// TwinCAT 3 PLC project PRG_MachineSystem
// ProgramVersion: 3.1.4024.0
// CompilerDefines: VISU_USEWSTRING
// libraries:
//   B_Base, * (RafalOS)
//   B_Base_HMI_Connector, * (RafalOS)
//   B_HMIManager, * (RafałOS)
//   B_MachineControl, * (RafalOS)
//   B_MachineControl_HMI_Connector, * (RafalOS)
//   B_MachineSystem, * (RafalOS)
//   B_PLCHMIManager, * (RafalOS)
//   Tc2_Standard, * (Beckhoff Automation GmbH)
//   Tc2_System, * (Beckhoff Automation GmbH)
//   Tc3_Module, * (Beckhoff Automation GmbH)
//   VisuSymbols,3.5.10.0,System
// project tree:
//   / DefaultInit.TcTTO, GlobalTextList.TcGTLO, MachineInit.TcTTO, PlcTask.TcTTO (not stored), Visualization Manager.TcVMO (not stored), VISU_TASK.TcTTO (not stored)
//   GVLs/ GVL_MachineVariable.TcGVL, GVL_TE1.TcGVL, GVL_TE2.TcGVL
//   POUs/01_MachineConfiguration/ FB_MachineConfiguration.TcPOU
//   POUs/02_HMIConfiguration/ FB_HMIConfiguration.TcPOU
//   POUs/03_CreatingTemplateRecipe/ FB_MachineTemplate1.TcPOU, FB_MachineTemplate2.TcPOU, FB_MachineTemplate3.TcPOU
//   POUs/04_TopElement1/3GE_B/ FB_GroupE_TE1.TcPOU, ITF_GroupE_TE1.TcIO, ITF_GroupE_TE1_HMI_Connector.TcIO, ITF_GroupE_TE1_HMI_Init.TcIO
//   POUs/04_TopElement1/3GE_B_HMI/ FB_GroupE_TE1_HMI.TcPOU, ITF_GroupE_TE1_HMI.TcIO, ST_GroupE_TE1_HMI.TcDUT, ST_GroupE_TE1_HMI_Link.TcDUT
//   POUs/04_TopElement1/9TE_B/ FB_TopElement1.TcPOU, ITF_TopElement1_HMI_Init.TcIO, ITF_TopElement1_HMI_Connector.TcIO, ITF_TopElement1.TcIO (not stored)
//   POUs/04_TopElement1/9TE_B_HMI/ FB_TopElement1_HMI.TcPOU, ITF_TopElement1_HMI.TcIO, ST_TopElement1_HMI.TcDUT, ST_TopElement1_HMI_Link.TcDUT
//   POUs/04_TopElement1/1C_B/ FB_Component_TE1.TcPOU, ITF_Component_TE1.TcIO, ITF_Component_TE1_HMI_Init.TcIO, ITF_Component_TE1_HMI_Connector.TcIO
//   POUs/04_TopElement1/2CE_B/ FB_ControlE_TE1.TcPOU, ITF_ControlE_TE1.TcIO, ITF_ControlE_TE1_HMI_Connector.TcIO, ITF_ControlE_TE1_HMI_Init.TcIO
//   POUs/04_TopElement1/1C_B_HMI/ FB_Component_TE1_HMI.TcPOU, ITF_Component_TE1_HMI.TcIO, ST_Component_TE1_HMI.TcDUT, ST_Component_TE1_HMI_Link.TcDUT
//   POUs/04_TopElement1/2CE_B_HMI/ FB_ControlE_TE1_HMI.TcPOU, ITF_ControlE_TE1_HMI.TcIO, ST_ControlE_TE1_HMI.TcDUT, ST_ControlE_TE1_HMI_Link.TcDUT
//   POUs/05_TopElement2/1C_B/ FB_Component_TE2.TcPOU, ITF_Component_TE2.TcIO, ITF_Component_TE2_HMI_Connector.TcIO, ITF_Component_TE2_HMI_Init.TcIO
//   POUs/05_TopElement2/1C_B_HMI/ FB_Component_TE2_HMI.TcPOU, ITF_Component_TE2_HMI.TcIO, ST_Component_TE2_HMI.TcDUT, ST_Component_TE2_HMI_Link.TcDUT
//   POUs/05_TopElement2/2CE_B/ FB_ControlE_TE2.TcPOU, ITF_ControlE_TE2.TcIO, ITF_ControlE_TE2_HMI_Connector.TcIO, ITF_ControlE_TE2_HMI_Init.TcIO
//   POUs/05_TopElement2/2CE_B_HMI/ FB_ControlE_TE2_HMI.TcPOU, ITF_ControlE_TE2_HMI.TcIO, ST_ControlE_TE2_HMI.TcDUT, ST_ControlE_TE2_HMI_Link.TcDUT
//   POUs/05_TopElement2/3GE_B/ FB_GroupE_TE2.TcPOU, ITF_GroupE_TE2.TcIO, ITF_GroupE_TE2_HMI_Connector.TcIO, ITF_GroupE_TE2_HMI_Init.TcIO
//   POUs/05_TopElement2/3GE_B_HMI/ FB_GroupE_TE2_HMI.TcPOU, ITF_GroupE_TE2_HMI.TcIO, ST_GroupE_TE2_HMI.TcDUT, ST_GroupE_TE2_HMI_Link.TcDUT
//   POUs/05_TopElement2/9TE_B/ FB_TopElement2.TcPOU, ITF_TopElement2.TcIO, ITF_TopElement2_HMI_Connector.TcIO, ITF_TopElement2_HMI_Init.TcIO
//   POUs/05_TopElement2/9TE_B_HMI/ FB_TopElement2_HMI.TcPOU, ITF_TopElement2_HMI.TcIO, ST_TopElement2_HMI.TcDUT, ST_TopElement2_HMI_Link.TcDUT
//   POUs/ PRG_MachineConfigure.TcPOU
//   VISUs/ MainScreen.TcVIS
// real-time tasks:
//   TASK PlcTask: cycle T#10ms, priority 10, ADS port 350
//   TASK VISU_TASK: cycle T#200000us, priority 12, ADS port 351
//   TASK DefaultInit: cycle T#10ms, priority 20, ADS port 352
//   TASK MachineInit: cycle T#10ms, priority 21, ADS port 353

CONFIGURATION PRG_MachineSystem
    RESOURCE PLC ON TwinCAT3
        TASK DefaultInit(INTERVAL := T#10ms, PRIORITY := 20);
        TASK MachineInit(INTERVAL := T#10ms, PRIORITY := 21);
        PROGRAM PRG_SystemControlMachineInit WITH DefaultInit : PRG_SystemControlMachineInit;
        PROGRAM PRG_ControlHMIInit WITH DefaultInit : PRG_ControlHMIInit;
        PROGRAM PRG_MachineConfigure WITH MachineInit : PRG_MachineConfigure;
    END_RESOURCE
END_CONFIGURATION

// ---- POUs/04_TopElement1/3GE_B_HMI/ST_GroupE_TE1_HMI.TcDUT
TYPE ST_GroupE_TE1_HMI :
STRUCT
	bZmienneTypoweDlaGE_TE1	: BOOL;
	
END_STRUCT
END_TYPE

// ---- POUs/04_TopElement1/3GE_B_HMI/ST_GroupE_TE1_HMI_Link.TcDUT
TYPE ST_GroupE_TE1_HMI_Link EXTENDS ST_BaseGroupElement_HMI_Link :
STRUCT
	stGroupE_TE1		: ST_GroupE_TE1_HMI;
	
	stControlE1_TE1		: ST_ControlE_TE1_HMI_Link;
	stControlE2_TE1		: ST_ControlE_TE1_HMI_Link;
	
	stComponetE1_TE1	: ST_Component_TE1_HMI_Link;
	stComponetE2_TE1	: ST_Component_TE1_HMI_Link;
	stComponetE3_TE1	: ST_Component_TE1_HMI_Link;
	stComponetE4_TE1	: ST_Component_TE1_HMI_Link;
	
END_STRUCT
END_TYPE

// ---- POUs/04_TopElement1/9TE_B_HMI/ST_TopElement1_HMI.TcDUT
TYPE ST_TopElement1_HMI :
STRUCT
	bZmienneTypoweDlaTopElement1	: BOOL;
	
END_STRUCT
END_TYPE

// ---- POUs/04_TopElement1/9TE_B_HMI/ST_TopElement1_HMI_Link.TcDUT
TYPE ST_TopElement1_HMI_Link EXTENDS ST_BaseTopElement_HMI_Link :
STRUCT
	stTopElement		: ST_TopElement1_HMI;
	
	stGE1				: ST_GroupE_TE1_HMI_Link;
	
	stCE1				: ST_ControlE_TE1_HMI_Link;
	stCE2				: ST_ControlE_TE1_HMI_Link;
	
	stC1				: ST_Component_TE1_HMI_Link;
	stC2				: ST_Component_TE1_HMI_Link;
	stC3				: ST_Component_TE1_HMI_Link;
	
END_STRUCT
END_TYPE

// ---- POUs/04_TopElement1/1C_B_HMI/ST_Component_TE1_HMI.TcDUT
TYPE ST_Component_TE1_HMI :
STRUCT
	bZmienneTypoweDlaComponent_TE1	: BOOL;
	
END_STRUCT
END_TYPE

// ---- POUs/04_TopElement1/1C_B_HMI/ST_Component_TE1_HMI_Link.TcDUT
TYPE ST_Component_TE1_HMI_Link EXTENDS ST_BaseComponent_HMI_Link :
STRUCT
	stComponent_TE1		: ST_Component_TE1_HMI;
	
	
END_STRUCT
END_TYPE

// ---- POUs/04_TopElement1/2CE_B_HMI/ST_ControlE_TE1_HMI.TcDUT
TYPE ST_ControlE_TE1_HMI :
STRUCT
	bZmienneTypoweDlaCE_TE1	: BOOL;
	
END_STRUCT
END_TYPE

// ---- POUs/04_TopElement1/2CE_B_HMI/ST_ControlE_TE1_HMI_Link.TcDUT
TYPE ST_ControlE_TE1_HMI_Link EXTENDS ST_BaseControlElement_HMI_Link :
STRUCT
	stControlE_TE1		: ST_ControlE_TE1_HMI;
	
	stComponetE1_TE1	: ST_Component_TE1_HMI_Link;
	stComponetE2_TE1	: ST_Component_TE1_HMI_Link;
	stComponetE3_TE1	: ST_Component_TE1_HMI_Link;
	stComponetE4_TE1	: ST_Component_TE1_HMI_Link;
	
END_STRUCT
END_TYPE

// ---- POUs/05_TopElement2/1C_B_HMI/ST_Component_TE2_HMI.TcDUT
TYPE ST_Component_TE2_HMI :
STRUCT
	bZmienneTypoweDlaComponent_TE2	: BOOL;
	
END_STRUCT
END_TYPE

// ---- POUs/05_TopElement2/1C_B_HMI/ST_Component_TE2_HMI_Link.TcDUT
TYPE ST_Component_TE2_HMI_Link EXTENDS ST_BaseComponent_HMI_Link :
STRUCT
	stComponent_TE2		: ST_Component_TE2_HMI;
	
	
END_STRUCT
END_TYPE

// ---- POUs/05_TopElement2/2CE_B_HMI/ST_ControlE_TE2_HMI.TcDUT
TYPE ST_ControlE_TE2_HMI :
STRUCT
	bZmienneTypoweDlaCE_TE2	: BOOL;
	
END_STRUCT
END_TYPE

// ---- POUs/05_TopElement2/2CE_B_HMI/ST_ControlE_TE2_HMI_Link.TcDUT
TYPE ST_ControlE_TE2_HMI_Link EXTENDS ST_BaseControlElement_HMI_Link :
STRUCT
	stControlE_TE2		: ST_ControlE_TE2_HMI;
	
	stComponetE1_TE2	: ST_Component_TE2_HMI_Link;
	stComponetE2_TE2	: ST_Component_TE2_HMI_Link;
	stComponetE3_TE2	: ST_Component_TE2_HMI_Link;
	stComponetE4_TE2	: ST_Component_TE2_HMI_Link;
	
END_STRUCT
END_TYPE

// ---- POUs/05_TopElement2/3GE_B_HMI/ST_GroupE_TE2_HMI.TcDUT
TYPE ST_GroupE_TE2_HMI :
STRUCT
	bZmienneTypoweDlaGE_TE2	: BOOL;
	
END_STRUCT
END_TYPE

// ---- POUs/05_TopElement2/3GE_B_HMI/ST_GroupE_TE2_HMI_Link.TcDUT
TYPE ST_GroupE_TE2_HMI_Link EXTENDS ST_BaseGroupElement_HMI_Link :
STRUCT
	stGroupE_TE2		: ST_GroupE_TE2_HMI;
	
	stControlE1_TE2		: ST_ControlE_TE2_HMI_Link;
	stControlE2_TE2		: ST_ControlE_TE2_HMI_Link;
	
	stComponetE1_TE2	: ST_Component_TE2_HMI_Link;
	stComponetE2_TE2	: ST_Component_TE2_HMI_Link;
	stComponetE3_TE2	: ST_Component_TE2_HMI_Link;
	stComponetE4_TE2	: ST_Component_TE2_HMI_Link;
	
END_STRUCT
END_TYPE

// ---- POUs/05_TopElement2/9TE_B_HMI/ST_TopElement2_HMI.TcDUT
TYPE ST_TopElement2_HMI :
STRUCT
	bZmienneTypoweDlaTopElement2	: BOOL;
	
END_STRUCT
END_TYPE

// ---- POUs/05_TopElement2/9TE_B_HMI/ST_TopElement2_HMI_Link.TcDUT
TYPE ST_TopElement2_HMI_Link EXTENDS ST_BaseTopElement_HMI_Link :
STRUCT
	stTopElement		: ST_TopElement2_HMI;
	
	stGE1				: ST_GroupE_TE2_HMI_Link;
	
	stCE1				: ST_ControlE_TE2_HMI_Link;
	stCE2				: ST_ControlE_TE2_HMI_Link;
	
	stC1				: ST_Component_TE2_HMI_Link;
	stC2				: ST_Component_TE2_HMI_Link;
	stC3				: ST_Component_TE2_HMI_Link;
	
END_STRUCT
END_TYPE

// ---- GVLs/GVL_MachineVariable.TcGVL
{attribute 'qualified_only'}
VAR_GLOBAL
	fbMachineConfiguration		: FB_MachineConfiguration;
	fbHMIConfiguration			: FB_HMIConfiguration;
	
	fbMachineTemplate1			: FB_MachineTemplate1;
	fbMachineTemplate2			: FB_MachineTemplate2;
	fbMachineTemplate3			: FB_MachineTemplate3;
	
END_VAR

// ---- GVLs/GVL_TE1.TcGVL
{attribute 'qualified_only'}
VAR_GLOBAL
(*	Control Element dla top element	*)
	fbComponent1CE1_TE1		: FB_Component_TE1;
	fbComponent2CE1_TE1		: FB_Component_TE1;
	fbComponent3CE1_TE1		: FB_Component_TE1;
	fbComponent4CE1_TE1		: FB_Component_TE1;
		
	fbControlE1_TE1			: FB_ControlE_TE1 (
								itfC1										:= fbComponent1CE1_TE1,
	                            itfC2										:= fbComponent2CE1_TE1,
	                            itfC3										:= fbComponent3CE1_TE1,
	                            itfC4										:= fbComponent4CE1_TE1
							);

	fbComponent1CE2_TE1		: FB_Component_TE1;
	fbComponent2CE2_TE1		: FB_Component_TE1;
	fbComponent3CE2_TE1		: FB_Component_TE1;
	fbComponent4CE2_TE1		: FB_Component_TE1;
		
	fbControlE2_TE1			: FB_ControlE_TE1 (
								itfC1										:= fbComponent1CE2_TE1,
	                            itfC2										:= fbComponent2CE2_TE1,
	                            itfC3										:= fbComponent3CE2_TE1,
	                            itfC4										:= fbComponent4CE2_TE1
							);
							
(*	element złożony	*)
	fbComponent1GE1_TE1			: FB_Component_TE1;
	fbComponent2GE1_TE1			: FB_Component_TE1;
	fbComponent3GE1_TE1			: FB_Component_TE1;
	fbComponent4GE1_TE1			: FB_Component_TE1;

	fbComponent1CE1GE1_TE1		: FB_Component_TE1;
	fbComponent2CE1GE1_TE1		: FB_Component_TE1;
	fbComponent3CE1GE1_TE1		: FB_Component_TE1;
	fbComponent4CE1GE1_TE1		: FB_Component_TE1;
		
	fbControlE1GE1_TE1			: FB_ControlE_TE1 (
								itfC1										:= fbComponent1CE1GE1_TE1,
	                            itfC2										:= fbComponent2CE1GE1_TE1,
	                            itfC3										:= fbComponent3CE1GE1_TE1,
	                            itfC4										:= fbComponent4CE1GE1_TE1
							);

	fbComponent1CE2GE1_TE1		: FB_Component_TE1;
	fbComponent2CE2GE1_TE1		: FB_Component_TE1;
	fbComponent3CE2GE1_TE1		: FB_Component_TE1;
	fbComponent4CE2GE1_TE1		: FB_Component_TE1;
		
	fbControlE2GE1_TE1			: FB_ControlE_TE1 (
								itfC1										:= fbComponent1CE2GE1_TE1,
	                            itfC2										:= fbComponent2CE2GE1_TE1,
	                            itfC3										:= fbComponent3CE2GE1_TE1,
	                            itfC4										:= fbComponent4CE2GE1_TE1
							);

	fbGroupE1_TE1			: FB_GroupE_TE1 (
								itfCE1										:= fbControlE1GE1_TE1,
	                            itfCE2										:= fbControlE2GE1_TE1,
	                            itfC1										:= fbComponent1GE1_TE1,
	                            itfC2										:= fbComponent2GE1_TE1,
	                            itfC3										:= fbComponent3GE1_TE1,
	                            itfC4										:= fbComponent4GE1_TE1
							);
							
							
(*	Komponenty TopElement1	*)
	fbComponent1_TE1		: FB_Component_TE1;
	fbComponent2_TE1		: FB_Component_TE1;
	fbComponent3_TE1		: FB_Component_TE1;
	
	fbTopElement1			: FB_TopElement1 (
								itfGE1										:= fbGroupE1_TE1,
								itfCE1										:= fbControlE1_TE1,
	                            itfCE2										:= fbControlE2_TE1,
								itfC1										:= fbComponent1_TE1,
								itfC2										:= fbComponent2_TE1,
								itfC3										:= fbComponent3_TE1
							);
	
(*	HMI	*)
	(* controlelementy *)
	fbComponent1CE1_TE1_HMI	: FB_Component_TE1_HMI (
								itfBaseLoggerConnector						:= GVL_SystemVariable.fbLogger,
	                            itfComponent_TE1Connector					:= fbComponent1CE1_TE1
							);
	fbComponent2CE1_TE1_HMI	: FB_Component_TE1_HMI (
								itfBaseLoggerConnector						:= GVL_SystemVariable.fbLogger,
	                            itfComponent_TE1Connector					:= fbComponent2CE1_TE1
							);
	fbComponent3CE1_TE1_HMI	: FB_Component_TE1_HMI (
								itfBaseLoggerConnector						:= GVL_SystemVariable.fbLogger,
	                            itfComponent_TE1Connector					:= fbComponent3CE1_TE1
							);
	fbComponent4CE1_TE1_HMI	: FB_Component_TE1_HMI (
								itfBaseLoggerConnector						:= GVL_SystemVariable.fbLogger,
	                            itfComponent_TE1Connector					:= fbComponent4CE1_TE1
							);

	fbControlE1_TE1_HMI			: FB_ControlE_TE1_HMI (
								itfBaseLoggerConnector						:= GVL_SystemVariable.fbLogger,
								itfControlE_TE1Connector					:= fbControlE1_TE1,
								itfC1										:= fbComponent1CE1_TE1_HMI,
	                            itfC2										:= fbComponent2CE1_TE1_HMI,
	                            itfC3										:= fbComponent3CE1_TE1_HMI,
	                            itfC4										:= fbComponent4CE1_TE1_HMI
							);

	fbComponent1CE2_TE1_HMI	: FB_Component_TE1_HMI (
								itfBaseLoggerConnector						:= GVL_SystemVariable.fbLogger,
	                            itfComponent_TE1Connector					:= fbComponent1CE2_TE1
							);
	fbComponent2CE2_TE1_HMI	: FB_Component_TE1_HMI (
								itfBaseLoggerConnector						:= GVL_SystemVariable.fbLogger,
	                            itfComponent_TE1Connector					:= fbComponent2CE2_TE1
							);
	fbComponent3CE2_TE1_HMI	: FB_Component_TE1_HMI (
								itfBaseLoggerConnector						:= GVL_SystemVariable.fbLogger,
	                            itfComponent_TE1Connector					:= fbComponent3CE2_TE1
							);
	fbComponent4CE2_TE1_HMI	: FB_Component_TE1_HMI (
								itfBaseLoggerConnector						:= GVL_SystemVariable.fbLogger,
	                            itfComponent_TE1Connector					:= fbComponent4CE2_TE1
							);

	fbControlE2_TE1_HMI			: FB_ControlE_TE1_HMI (
								itfBaseLoggerConnector						:= GVL_SystemVariable.fbLogger,
								itfControlE_TE1Connector					:= fbControlE2_TE1,
								itfC1										:= fbComponent1CE2_TE1_HMI,
	                            itfC2										:= fbComponent2CE2_TE1_HMI,
	                            itfC3										:= fbComponent3CE2_TE1_HMI,
	                            itfC4										:= fbComponent4CE2_TE1_HMI
							);
							
	(*	group element 	*)
	fbComponent1GE1_TE1_HMI	: FB_Component_TE1_HMI (
								itfBaseLoggerConnector						:= GVL_SystemVariable.fbLogger,
	                            itfComponent_TE1Connector					:= fbComponent1GE1_TE1
							);
	fbComponent2GE1_TE1_HMI	: FB_Component_TE1_HMI (
								itfBaseLoggerConnector						:= GVL_SystemVariable.fbLogger,
	                            itfComponent_TE1Connector					:= fbComponent2GE1_TE1
							);
	fbComponent3GE1_TE1_HMI	: FB_Component_TE1_HMI (
								itfBaseLoggerConnector						:= GVL_SystemVariable.fbLogger,
	                            itfComponent_TE1Connector					:= fbComponent3GE1_TE1
							);
	fbComponent4GE1_TE1_HMI	: FB_Component_TE1_HMI (
								itfBaseLoggerConnector						:= GVL_SystemVariable.fbLogger,
	                            itfComponent_TE1Connector					:= fbComponent4GE1_TE1
							);

	
	
	fbComponent1CE1GE1_TE1_HMI	: FB_Component_TE1_HMI (
								itfBaseLoggerConnector						:= GVL_SystemVariable.fbLogger,
	                            itfComponent_TE1Connector					:= fbComponent1CE1GE1_TE1
							);
	fbComponent2CE1GE1_TE1_HMI	: FB_Component_TE1_HMI (
								itfBaseLoggerConnector						:= GVL_SystemVariable.fbLogger,
	                            itfComponent_TE1Connector					:= fbComponent2CE1GE1_TE1
							);
	fbComponent3CE1GE1_TE1_HMI	: FB_Component_TE1_HMI (
								itfBaseLoggerConnector						:= GVL_SystemVariable.fbLogger,
	                            itfComponent_TE1Connector					:= fbComponent3CE1GE1_TE1
							);
	fbComponent4CE1GE1_TE1_HMI	: FB_Component_TE1_HMI (
								itfBaseLoggerConnector						:= GVL_SystemVariable.fbLogger,
	                            itfComponent_TE1Connector					:= fbComponent4CE1GE1_TE1
							);

	fbControlE1GE1_TE1_HMI	: FB_ControlE_TE1_HMI (
								itfBaseLoggerConnector						:= GVL_SystemVariable.fbLogger,
								itfControlE_TE1Connector					:= fbControlE1GE1_TE1,
								itfC1										:= fbComponent1CE1GE1_TE1_HMI,
	                            itfC2										:= fbComponent2CE1GE1_TE1_HMI,
	                            itfC3										:= fbComponent3CE1GE1_TE1_HMI,
	                            itfC4										:= fbComponent4CE1GE1_TE1_HMI
							);

	fbComponent1CE2GE1_TE1_HMI	: FB_Component_TE1_HMI (
								itfBaseLoggerConnector						:= GVL_SystemVariable.fbLogger,
	                            itfComponent_TE1Connector					:= fbComponent1CE2GE1_TE1
							);
	fbComponent2CE2GE1_TE1_HMI	: FB_Component_TE1_HMI (
								itfBaseLoggerConnector						:= GVL_SystemVariable.fbLogger,
	                            itfComponent_TE1Connector					:= fbComponent2CE2GE1_TE1
							);
	fbComponent3CE2GE1_TE1_HMI	: FB_Component_TE1_HMI (
								itfBaseLoggerConnector						:= GVL_SystemVariable.fbLogger,
	                            itfComponent_TE1Connector					:= fbComponent3CE2GE1_TE1
							);
	fbComponent4CE2GE1_TE1_HMI	: FB_Component_TE1_HMI (
								itfBaseLoggerConnector						:= GVL_SystemVariable.fbLogger,
	                            itfComponent_TE1Connector					:= fbComponent4CE2GE1_TE1
							);

	fbControlE2GE1_TE1_HMI	: FB_ControlE_TE1_HMI (
								itfBaseLoggerConnector						:= GVL_SystemVariable.fbLogger,
								itfControlE_TE1Connector					:= fbControlE2GE1_TE1,
								itfC1										:= fbComponent1CE2GE1_TE1_HMI,
	                            itfC2										:= fbComponent2CE2GE1_TE1_HMI,
	                            itfC3										:= fbComponent3CE2GE1_TE1_HMI,
	                            itfC4										:= fbComponent4CE2GE1_TE1_HMI
							);						
	fbGroupE1_TE1_HMI		: FB_GroupE_TE1_HMI (
								itfBaseLoggerConnector						:= GVL_SystemVariable.fbLogger,
	                            itfGroupE_TE1Connector						:= fbGroupE1_TE1,
	                            itfCE1										:= fbControlE1GE1_TE1_HMI,
	                            itfCE2										:= fbControlE2GE1_TE1_HMI,
	                            itfC1										:= fbComponent1GE1_TE1_HMI,
	                            itfC2										:= fbComponent2GE1_TE1_HMI,
	                            itfC3										:= fbComponent3GE1_TE1_HMI,
	                            itfC4										:= fbComponent4GE1_TE1_HMI
	
							);
	
	(* komponenty te	*)
	fbComponent1_TE1_HMI	: FB_Component_TE1_HMI (
								itfBaseLoggerConnector						:= GVL_SystemVariable.fbLogger,
	                            itfComponent_TE1Connector					:= fbComponent1_TE1
							);
	fbComponent2_TE1_HMI	: FB_Component_TE1_HMI (
								itfBaseLoggerConnector						:= GVL_SystemVariable.fbLogger,
	                            itfComponent_TE1Connector					:= fbComponent2_TE1
							);
	fbComponent3_TE1_HMI	: FB_Component_TE1_HMI (
								itfBaseLoggerConnector						:= GVL_SystemVariable.fbLogger,
	                            itfComponent_TE1Connector					:= fbComponent3_TE1
							);
	

	fbTopElement1HMI		: FB_TopElement1_HMI (
										itfBaseLoggerConnector				:= GVL_SystemVariable.fbLogger,
                                        itfTopElementConnector				:= fbTopElement1,
										itfGE1								:= fbGroupE1_TE1_HMI,
										itfCE1								:= fbControlE1_TE1_HMI,
		    	                        itfCE2								:= fbControlE2_TE1_HMI,
										itfC1								:= fbComponent1_TE1_HMI,
										itfC2								:= fbComponent2_TE1_HMI,
										itfC3								:= fbComponent3_TE1_HMI
							);
	stTopElemenent1			: ST_TopElement1_HMI_Link;
							
END_VAR

// ---- GVLs/GVL_TE2.TcGVL
{attribute 'qualified_only'}
VAR_GLOBAL
(*	Control Element dla top element	*)
	fbComponent1CE1_TE2		: FB_Component_TE2;
	fbComponent2CE1_TE2		: FB_Component_TE2;
	fbComponent3CE1_TE2		: FB_Component_TE2;
	fbComponent4CE1_TE2		: FB_Component_TE2;
		
	fbControlE1_TE2			: FB_ControlE_TE2 (
								itfC1										:= fbComponent1CE1_TE2,
	                            itfC2										:= fbComponent2CE1_TE2,
	                            itfC3										:= fbComponent3CE1_TE2,
	                            itfC4										:= fbComponent4CE1_TE2
							);

	fbComponent1CE2_TE2		: FB_Component_TE2;
	fbComponent2CE2_TE2		: FB_Component_TE2;
	fbComponent3CE2_TE2		: FB_Component_TE2;
	fbComponent4CE2_TE2		: FB_Component_TE2;
		
	fbControlE2_TE2			: FB_ControlE_TE2 (
								itfC1										:= fbComponent1CE2_TE2,
	                            itfC2										:= fbComponent2CE2_TE2,
	                            itfC3										:= fbComponent3CE2_TE2,
	                            itfC4										:= fbComponent4CE2_TE2
							);
							
(*	element złożony	*)
	fbComponent1GE1_TE2			: FB_Component_TE2;
	fbComponent2GE1_TE2			: FB_Component_TE2;
	fbComponent3GE1_TE2			: FB_Component_TE2;
	fbComponent4GE1_TE2			: FB_Component_TE2;

	fbComponent1CE1GE1_TE2		: FB_Component_TE2;
	fbComponent2CE1GE1_TE2		: FB_Component_TE2;
	fbComponent3CE1GE1_TE2		: FB_Component_TE2;
	fbComponent4CE1GE1_TE2		: FB_Component_TE2;
		
	fbControlE1GE1_TE2			: FB_ControlE_TE2 (
								itfC1										:= fbComponent1CE1GE1_TE2,
	                            itfC2										:= fbComponent2CE1GE1_TE2,
	                            itfC3										:= fbComponent3CE1GE1_TE2,
	                            itfC4										:= fbComponent4CE1GE1_TE2
							);

	fbComponent1CE2GE1_TE2		: FB_Component_TE2;
	fbComponent2CE2GE1_TE2		: FB_Component_TE2;
	fbComponent3CE2GE1_TE2		: FB_Component_TE2;
	fbComponent4CE2GE1_TE2		: FB_Component_TE2;
		
	fbControlE2GE1_TE2			: FB_ControlE_TE2 (
								itfC1										:= fbComponent1CE2GE1_TE2,
	                            itfC2										:= fbComponent2CE2GE1_TE2,
	                            itfC3										:= fbComponent3CE2GE1_TE2,
	                            itfC4										:= fbComponent4CE2GE1_TE2
							);

	fbGroupE1_TE2			: FB_GroupE_TE2 (
								itfCE1										:= fbControlE1GE1_TE2,
	                            itfCE2										:= fbControlE2GE1_TE2,
	                            itfC1										:= fbComponent1GE1_TE2,
	                            itfC2										:= fbComponent2GE1_TE2,
	                            itfC3										:= fbComponent3GE1_TE2,
	                            itfC4										:= fbComponent4GE1_TE2
							);
							
							
(*	Komponenty TopElement1	*)
	fbComponent1_TE2		: FB_Component_TE2;
	fbComponent2_TE2		: FB_Component_TE2;
	fbComponent3_TE2		: FB_Component_TE2;
	
	fbTopElement2			: FB_TopElement2 (
								itfGE1										:= fbGroupE1_TE2,
								itfCE1										:= fbControlE1_TE2,
	                            itfCE2										:= fbControlE2_TE2,
								itfC1										:= fbComponent1_TE2,
								itfC2										:= fbComponent2_TE2,
								itfC3										:= fbComponent3_TE2
							);
	
(*	HMI	*)
	(* controlelementy *)
	fbComponent1CE1_TE2_HMI	: FB_Component_TE2_HMI (
								itfBaseLoggerConnector						:= GVL_SystemVariable.fbLogger,
	                            itfComponent_TE2Connector					:= fbComponent1CE1_TE2
							);
	fbComponent2CE1_TE2_HMI	: FB_Component_TE2_HMI (
								itfBaseLoggerConnector						:= GVL_SystemVariable.fbLogger,
	                            itfComponent_TE2Connector					:= fbComponent2CE1_TE2
							);
	fbComponent3CE1_TE2_HMI	: FB_Component_TE2_HMI (
								itfBaseLoggerConnector						:= GVL_SystemVariable.fbLogger,
	                            itfComponent_TE2Connector					:= fbComponent3CE1_TE2
							);
	fbComponent4CE1_TE2_HMI	: FB_Component_TE2_HMI (
								itfBaseLoggerConnector						:= GVL_SystemVariable.fbLogger,
	                            itfComponent_TE2Connector					:= fbComponent4CE1_TE2
							);

	fbControlE1_TE2_HMI			: FB_ControlE_TE2_HMI (
								itfBaseLoggerConnector						:= GVL_SystemVariable.fbLogger,
								itfControlE_TE2Connector					:= fbControlE1_TE2,
								itfC1										:= fbComponent1CE1_TE2_HMI,
	                            itfC2										:= fbComponent2CE1_TE2_HMI,
	                            itfC3										:= fbComponent3CE1_TE2_HMI,
	                            itfC4										:= fbComponent4CE1_TE2_HMI
							);

	fbComponent1CE2_TE2_HMI	: FB_Component_TE2_HMI (
								itfBaseLoggerConnector						:= GVL_SystemVariable.fbLogger,
	                            itfComponent_TE2Connector					:= fbComponent1CE2_TE2
							);
	fbComponent2CE2_TE2_HMI	: FB_Component_TE2_HMI (
								itfBaseLoggerConnector						:= GVL_SystemVariable.fbLogger,
	                            itfComponent_TE2Connector					:= fbComponent2CE2_TE2
							);
	fbComponent3CE2_TE2_HMI	: FB_Component_TE2_HMI (
								itfBaseLoggerConnector						:= GVL_SystemVariable.fbLogger,
	                            itfComponent_TE2Connector					:= fbComponent3CE2_TE2
							);
	fbComponent4CE2_TE2_HMI	: FB_Component_TE2_HMI (
								itfBaseLoggerConnector						:= GVL_SystemVariable.fbLogger,
	                            itfComponent_TE2Connector					:= fbComponent4CE2_TE2
							);

	fbControlE2_TE2_HMI			: FB_ControlE_TE2_HMI (
								itfBaseLoggerConnector						:= GVL_SystemVariable.fbLogger,
								itfControlE_TE2Connector					:= fbControlE2_TE2,
								itfC1										:= fbComponent1CE2_TE2_HMI,
	                            itfC2										:= fbComponent2CE2_TE2_HMI,
	                            itfC3										:= fbComponent3CE2_TE2_HMI,
	                            itfC4										:= fbComponent4CE2_TE2_HMI
							);
							
	(*	group element 	*)
	fbComponent1GE1_TE2_HMI	: FB_Component_TE2_HMI (
								itfBaseLoggerConnector						:= GVL_SystemVariable.fbLogger,
	                            itfComponent_TE2Connector					:= fbComponent1GE1_TE2
							);
	fbComponent2GE1_TE2_HMI	: FB_Component_TE2_HMI (
								itfBaseLoggerConnector						:= GVL_SystemVariable.fbLogger,
	                            itfComponent_TE2Connector					:= fbComponent2GE1_TE2
							);
	fbComponent3GE1_TE2_HMI	: FB_Component_TE2_HMI (
								itfBaseLoggerConnector						:= GVL_SystemVariable.fbLogger,
	                            itfComponent_TE2Connector					:= fbComponent3GE1_TE2
							);
	fbComponent4GE1_TE2_HMI	: FB_Component_TE2_HMI (
								itfBaseLoggerConnector						:= GVL_SystemVariable.fbLogger,
	                            itfComponent_TE2Connector					:= fbComponent4GE1_TE2
							);

	
	
	fbComponent1CE1GE1_TE2_HMI	: FB_Component_TE2_HMI (
								itfBaseLoggerConnector						:= GVL_SystemVariable.fbLogger,
	                            itfComponent_TE2Connector					:= fbComponent1CE1GE1_TE2
							);
	fbComponent2CE1GE1_TE2_HMI	: FB_Component_TE2_HMI (
								itfBaseLoggerConnector						:= GVL_SystemVariable.fbLogger,
	                            itfComponent_TE2Connector					:= fbComponent2CE1GE1_TE2
							);
	fbComponent3CE1GE1_TE2_HMI	: FB_Component_TE2_HMI (
								itfBaseLoggerConnector						:= GVL_SystemVariable.fbLogger,
	                            itfComponent_TE2Connector					:= fbComponent3CE1GE1_TE2
							);
	fbComponent4CE1GE1_TE2_HMI	: FB_Component_TE2_HMI (
								itfBaseLoggerConnector						:= GVL_SystemVariable.fbLogger,
	                            itfComponent_TE2Connector					:= fbComponent4CE1GE1_TE2
							);

	fbControlE1GE1_TE2_HMI	: FB_ControlE_TE2_HMI (
								itfBaseLoggerConnector						:= GVL_SystemVariable.fbLogger,
								itfControlE_TE2Connector					:= fbControlE1GE1_TE2,
								itfC1										:= fbComponent1CE1GE1_TE2_HMI,
	                            itfC2										:= fbComponent2CE1GE1_TE2_HMI,
	                            itfC3										:= fbComponent3CE1GE1_TE2_HMI,
	                            itfC4										:= fbComponent4CE1GE1_TE2_HMI
							);

	fbComponent1CE2GE1_TE2_HMI	: FB_Component_TE2_HMI (
								itfBaseLoggerConnector						:= GVL_SystemVariable.fbLogger,
	                            itfComponent_TE2Connector					:= fbComponent1CE2GE1_TE2
							);
	fbComponent2CE2GE1_TE2_HMI	: FB_Component_TE2_HMI (
								itfBaseLoggerConnector						:= GVL_SystemVariable.fbLogger,
	                            itfComponent_TE2Connector					:= fbComponent2CE2GE1_TE2
							);
	fbComponent3CE2GE1_TE2_HMI	: FB_Component_TE2_HMI (
								itfBaseLoggerConnector						:= GVL_SystemVariable.fbLogger,
	                            itfComponent_TE2Connector					:= fbComponent3CE2GE1_TE2
							);
	fbComponent4CE2GE1_TE2_HMI	: FB_Component_TE2_HMI (
								itfBaseLoggerConnector						:= GVL_SystemVariable.fbLogger,
	                            itfComponent_TE2Connector					:= fbComponent4CE2GE1_TE2
							);

	fbControlE2GE1_TE2_HMI	: FB_ControlE_TE2_HMI (
								itfBaseLoggerConnector						:= GVL_SystemVariable.fbLogger,
								itfControlE_TE2Connector					:= fbControlE2GE1_TE2,
								itfC1										:= fbComponent1CE2GE1_TE2_HMI,
	                            itfC2										:= fbComponent2CE2GE1_TE2_HMI,
	                            itfC3										:= fbComponent3CE2GE1_TE2_HMI,
	                            itfC4										:= fbComponent4CE2GE1_TE2_HMI
							);						
	fbGroupE1_TE2_HMI		: FB_GroupE_TE2_HMI (
								itfBaseLoggerConnector						:= GVL_SystemVariable.fbLogger,
	                            itfGroupE_TE2Connector						:= fbGroupE1_TE2,
	                            itfCE1										:= fbControlE1GE1_TE2_HMI,
	                            itfCE2										:= fbControlE2GE1_TE2_HMI,
	                            itfC1										:= fbComponent1GE1_TE2_HMI,
	                            itfC2										:= fbComponent2GE1_TE2_HMI,
	                            itfC3										:= fbComponent3GE1_TE2_HMI,
	                            itfC4										:= fbComponent4GE1_TE2_HMI
	
							);
	
	(* komponenty te	*)
	fbComponent1_TE2_HMI	: FB_Component_TE2_HMI (
								itfBaseLoggerConnector						:= GVL_SystemVariable.fbLogger,
	                            itfComponent_TE2Connector					:= fbComponent1_TE2
							);
	fbComponent2_TE2_HMI	: FB_Component_TE2_HMI (
								itfBaseLoggerConnector						:= GVL_SystemVariable.fbLogger,
	                            itfComponent_TE2Connector					:= fbComponent2_TE2
							);
	fbComponent3_TE2_HMI	: FB_Component_TE2_HMI (
								itfBaseLoggerConnector						:= GVL_SystemVariable.fbLogger,
	                            itfComponent_TE2Connector					:= fbComponent3_TE2
							);
	

	fbTopElement2HMI		: FB_TopElement2_HMI (
										itfBaseLoggerConnector				:= GVL_SystemVariable.fbLogger,
                                        itfTopElementConnector				:= fbTopElement2,
										itfGE1								:= fbGroupE1_TE2_HMI,
										itfCE1								:= fbControlE1_TE2_HMI,
		    	                        itfCE2								:= fbControlE2_TE2_HMI,
										itfC1								:= fbComponent1_TE2_HMI,
										itfC2								:= fbComponent2_TE2_HMI,
										itfC3								:= fbComponent3_TE2_HMI
							);
	stTopElemenent2			: ST_TopElement2_HMI_Link;
							
END_VAR

// ---- POUs/04_TopElement1/3GE_B/ITF_GroupE_TE1.TcIO
INTERFACE ITF_GroupE_TE1 EXTENDS ITF_BaseGroupElement

METHOD testMethodGE : BOOL
VAR_INPUT
END_VAR
END_METHOD

END_INTERFACE

// ---- POUs/04_TopElement1/3GE_B/ITF_GroupE_TE1_HMI_Connector.TcIO
INTERFACE ITF_GroupE_TE1_HMI_Connector EXTENDS ITF_BaseGroupElement_HMI_Connector

END_INTERFACE

// ---- POUs/04_TopElement1/3GE_B/ITF_GroupE_TE1_HMI_Init.TcIO
INTERFACE ITF_GroupE_TE1_HMI_Init EXTENDS ITF_BaseGroupElement, ITF_GroupE_TE1_HMI_Connector

END_INTERFACE

// ---- POUs/04_TopElement1/3GE_B_HMI/ITF_GroupE_TE1_HMI.TcIO
INTERFACE ITF_GroupE_TE1_HMI EXTENDS ITF_BaseGroupElement_HMI

METHOD LinkGroupEData : BOOL
VAR_INPUT
	stData				: REFERENCE TO ST_GroupE_TE1_HMI_Link;
END_VAR
END_METHOD

END_INTERFACE

// ---- POUs/04_TopElement1/9TE_B/ITF_TopElement1_HMI_Init.TcIO
INTERFACE ITF_TopElement1_HMI_Init EXTENDS ITF_BaseTopElement, ITF_TopElement1_HMI_Connector

END_INTERFACE

// ---- POUs/04_TopElement1/9TE_B/ITF_TopElement1_HMI_Connector.TcIO
INTERFACE ITF_TopElement1_HMI_Connector EXTENDS ITF_BaseTopElement_HMI_Connector

END_INTERFACE

// ---- POUs/04_TopElement1/9TE_B_HMI/ITF_TopElement1_HMI.TcIO
INTERFACE ITF_TopElement1_HMI EXTENDS ITF_BaseTopElement_HMI

END_INTERFACE

// ---- POUs/04_TopElement1/1C_B/ITF_Component_TE1.TcIO
INTERFACE ITF_Component_TE1 EXTENDS ITF_BaseComponent

METHOD testMethod : BOOL
VAR_INPUT
END_VAR
END_METHOD

END_INTERFACE

// ---- POUs/04_TopElement1/1C_B/ITF_Component_TE1_HMI_Init.TcIO
INTERFACE ITF_Component_TE1_HMI_Init EXTENDS ITF_BaseComponent, ITF_Component_TE1_HMI_Connector

END_INTERFACE

// ---- POUs/04_TopElement1/1C_B/ITF_Component_TE1_HMI_Connector.TcIO
INTERFACE ITF_Component_TE1_HMI_Connector EXTENDS ITF_BaseComponent_HMI_Connector

END_INTERFACE

// ---- POUs/04_TopElement1/2CE_B/ITF_ControlE_TE1.TcIO
INTERFACE ITF_ControlE_TE1 EXTENDS ITF_BaseControlElement

METHOD testMethodCE : BOOL
VAR_INPUT
END_VAR
END_METHOD

END_INTERFACE

// ---- POUs/04_TopElement1/2CE_B/ITF_ControlE_TE1_HMI_Connector.TcIO
INTERFACE ITF_ControlE_TE1_HMI_Connector EXTENDS ITF_BaseControlElement_HMI_Connector

END_INTERFACE

// ---- POUs/04_TopElement1/2CE_B/ITF_ControlE_TE1_HMI_Init.TcIO
INTERFACE ITF_ControlE_TE1_HMI_Init EXTENDS ITF_BaseControlElement, ITF_ControlE_TE1_HMI_Connector

END_INTERFACE

// ---- POUs/04_TopElement1/1C_B_HMI/ITF_Component_TE1_HMI.TcIO
INTERFACE ITF_Component_TE1_HMI EXTENDS ITF_BaseComponent_HMI

METHOD LinkComponentData : BOOL
VAR_INPUT
	stData				: REFERENCE TO ST_Component_TE1_HMI_Link;
END_VAR
END_METHOD

END_INTERFACE

// ---- POUs/04_TopElement1/2CE_B_HMI/ITF_ControlE_TE1_HMI.TcIO
INTERFACE ITF_ControlE_TE1_HMI EXTENDS ITF_BaseControlElement_HMI

METHOD LinkControlEData : BOOL
VAR_INPUT
	stData				: REFERENCE TO ST_ControlE_TE1_HMI_Link;
END_VAR
END_METHOD

END_INTERFACE

// ---- POUs/05_TopElement2/1C_B/ITF_Component_TE2.TcIO
INTERFACE ITF_Component_TE2 EXTENDS ITF_BaseComponent

METHOD testMethod : BOOL
VAR_INPUT
END_VAR
END_METHOD

END_INTERFACE

// ---- POUs/05_TopElement2/1C_B/ITF_Component_TE2_HMI_Connector.TcIO
INTERFACE ITF_Component_TE2_HMI_Connector EXTENDS ITF_BaseComponent_HMI_Connector

END_INTERFACE

// ---- POUs/05_TopElement2/1C_B/ITF_Component_TE2_HMI_Init.TcIO
INTERFACE ITF_Component_TE2_HMI_Init EXTENDS ITF_BaseComponent, ITF_Component_TE2_HMI_Connector

END_INTERFACE

// ---- POUs/05_TopElement2/1C_B_HMI/ITF_Component_TE2_HMI.TcIO
INTERFACE ITF_Component_TE2_HMI EXTENDS ITF_BaseComponent_HMI

METHOD LinkComponentData : BOOL
VAR_INPUT
	stData				: REFERENCE TO ST_Component_TE2_HMI_Link;
END_VAR
END_METHOD

END_INTERFACE

// ---- POUs/05_TopElement2/2CE_B/ITF_ControlE_TE2.TcIO
INTERFACE ITF_ControlE_TE2 EXTENDS ITF_BaseControlElement

METHOD testMethodCE : BOOL
VAR_INPUT
END_VAR
END_METHOD

END_INTERFACE

// ---- POUs/05_TopElement2/2CE_B/ITF_ControlE_TE2_HMI_Connector.TcIO
INTERFACE ITF_ControlE_TE2_HMI_Connector EXTENDS ITF_BaseControlElement_HMI_Connector

END_INTERFACE

// ---- POUs/05_TopElement2/2CE_B/ITF_ControlE_TE2_HMI_Init.TcIO
INTERFACE ITF_ControlE_TE2_HMI_Init EXTENDS ITF_BaseControlElement, ITF_ControlE_TE2_HMI_Connector

END_INTERFACE

// ---- POUs/05_TopElement2/2CE_B_HMI/ITF_ControlE_TE2_HMI.TcIO
INTERFACE ITF_ControlE_TE2_HMI EXTENDS ITF_BaseControlElement_HMI

METHOD LinkControlEData : BOOL
VAR_INPUT
	stData				: REFERENCE TO ST_ControlE_TE2_HMI_Link;
END_VAR
END_METHOD

END_INTERFACE

// ---- POUs/05_TopElement2/3GE_B/ITF_GroupE_TE2.TcIO
INTERFACE ITF_GroupE_TE2 EXTENDS ITF_BaseGroupElement

METHOD testMethodGE : BOOL
VAR_INPUT
END_VAR
END_METHOD

END_INTERFACE

// ---- POUs/05_TopElement2/3GE_B/ITF_GroupE_TE2_HMI_Connector.TcIO
INTERFACE ITF_GroupE_TE2_HMI_Connector EXTENDS ITF_BaseGroupElement_HMI_Connector

END_INTERFACE

// ---- POUs/05_TopElement2/3GE_B/ITF_GroupE_TE2_HMI_Init.TcIO
INTERFACE ITF_GroupE_TE2_HMI_Init EXTENDS ITF_BaseGroupElement, ITF_GroupE_TE2_HMI_Connector

END_INTERFACE

// ---- POUs/05_TopElement2/3GE_B_HMI/ITF_GroupE_TE2_HMI.TcIO
INTERFACE ITF_GroupE_TE2_HMI EXTENDS ITF_BaseGroupElement_HMI

METHOD LinkGroupEData : BOOL
VAR_INPUT
	stData				: REFERENCE TO ST_GroupE_TE2_HMI_Link;
END_VAR
END_METHOD

END_INTERFACE

// ---- POUs/05_TopElement2/9TE_B/ITF_TopElement2.TcIO
INTERFACE ITF_TopElement2

END_INTERFACE

// ---- POUs/05_TopElement2/9TE_B/ITF_TopElement2_HMI_Connector.TcIO
INTERFACE ITF_TopElement2_HMI_Connector EXTENDS ITF_BaseTopElement_HMI_Connector

END_INTERFACE

// ---- POUs/05_TopElement2/9TE_B/ITF_TopElement2_HMI_Init.TcIO
INTERFACE ITF_TopElement2_HMI_Init EXTENDS ITF_BaseTopElement, ITF_TopElement2_HMI_Connector

END_INTERFACE

// ---- POUs/05_TopElement2/9TE_B_HMI/ITF_TopElement2_HMI.TcIO
INTERFACE ITF_TopElement2_HMI EXTENDS ITF_BaseTopElement_HMI

END_INTERFACE

// ---- POUs/PRG_MachineConfigure.TcPOU
PROGRAM PRG_MachineConfigure
VAR
END_VAR

IF (NOT GVL_SystemVariable.bMachineInitDone) THEN

	PRG_SystemControlMachineInit.fbMachineConfigure.AddConfiguration (fbConfigure := GVL_MachineVariable.fbMachineConfiguration);
	PRG_ControlHMIInit.fbHMIConfigure.AddConfiguration (fbConfigure := GVL_MachineVariable.fbHMIConfiguration);
	
	GVL_SystemVariable.bMachineInitDone		:= TRUE;
END_IF

END_PROGRAM

// ---- POUs/01_MachineConfiguration/FB_MachineConfiguration.TcPOU
(*			
	RafalOS
	Rafał Osajda		10.11.2025		TC 4024.66
	Główny blok konfiguracyjny MachineControl
*)
FUNCTION_BLOCK FB_MachineConfiguration EXTENDS FB_Base IMPLEMENTS ITF_MCConfiguration
VAR

END_VAR

(*			
	RafalOS
	Rafał Osajda		26.11.2025		TC 4024.66
	Dodawanie szablonu receptury
*)
METHOD AddCreateTemplate : BOOL
VAR_INPUT
	itfMachineControl	: B_MachineControl.ITF_MCMachineControlConfigure;
END_VAR
itfMachineControl.AddCreateTemplateFromConfiguration (
	fbCreateTemplate := GVL_MachineVariable.fbMachineTemplate1
);
itfMachineControl.AddCreateTemplateFromConfiguration (
	fbCreateTemplate := GVL_MachineVariable.fbMachineTemplate2
);
itfMachineControl.AddCreateTemplateFromConfiguration (
	fbCreateTemplate := GVL_MachineVariable.fbMachineTemplate3
);
END_METHOD

(*			
	RafalOS
	Rafał Osajda		13.11.2025		TC 4024.66
	Metoda przeznaczona do dodawania elementów do FB_MachineControl
*)
METHOD AddElements : BOOL
VAR_INPUT
	itfMachineControl	: B_MachineControl.ITF_MCMachineControlConfigure;
END_VAR
THIS^.SetText (eLocation := E_BaseLocation.pl, wsDescription := "TopElement 1");
THIS^.SetText (eLocation := E_BaseLocation.en, wsDescription := "TopElement 1");
THIS^.SetText (eLocation := E_BaseLocation.de, wsDescription := "TopElement 1");
GVL_TE1.fbTopElement1.SetName (stName := THIS^.GetTexts ());
itfMachineControl.AddElementFromConfiguration (itfElements := GVL_TE1.fbTopElement1);

THIS^.SetText (eLocation := E_BaseLocation.pl, wsDescription := "TopElement 2");
THIS^.SetText (eLocation := E_BaseLocation.en, wsDescription := "TopElement 2");
THIS^.SetText (eLocation := E_BaseLocation.de, wsDescription := "TopElement 2");
GVL_TE2.fbTopElement2.SetName (stName := THIS^.GetTexts ());
itfMachineControl.AddElementFromConfiguration (itfElements := GVL_TE2.fbTopElement2);
END_METHOD

(*			
	RafalOS
	Rafał Osajda		13.11.2025		TC 4024.66
	Podpięcie menadżera HMI
*)
METHOD AddHMIManager : BOOL
VAR_INPUT
	itfMachineControl	: B_MachineControl.ITF_MCMachineControlConfigure;
END_VAR
END_METHOD

(*
	RafalOS
	Rafał Osajda		13.11.2025		TC 4024.66
	Dodanie samego siebie do systemu controli maszyny
*)
METHOD AddMachineCotrolToYourSelf : BOOL
VAR_INPUT
	itfMachineControl	: B_MachineControl.ITF_MCMachineControlConfigure;
END_VAR
END_METHOD

(*			
	RafalOS
	Rafał Osajda		26.11.2025		TC 4024.66
	Dodanie obsługi receptur
*)
METHOD AddModulRecipe : BOOL
VAR_INPUT
	itfMachineControl	: B_MachineControl.ITF_MCMachineControlConfigure;
END_VAR
END_METHOD

(*
	RafalOS
	Rafał Osajda		13.11.2025		TC 4024.66
	Dodanie modułu sterowania stanami i trybami do machinecontrol
*)
METHOD AddSaMCotrollerToMachineControl : BOOL
VAR_INPUT
	itfMachineControl	: B_MachineControl.ITF_MCMachineControlConfigure;
END_VAR
END_METHOD

METHOD AddSaMToTopElement
VAR_INPUT
	itfMachineControl	: B_MachineControl.ITF_MCMachineControlConfigure;
END_VAR
END_METHOD

(*			
	RafalOS
	Rafał Osajda		13.11.2025		TC 4024.66
	Zlinkowanie danych wspólnych do dodanych elementów
*)
METHOD LinkCommonDataToAddedElements : BOOL
VAR_INPUT
	itfMachineControl	: B_MachineControl.ITF_MCMachineControlConfigure;
END_VAR
END_METHOD

(*			
	RafalOS
	Rafał Osajda		13.11.2025		TC 4024.66
	Dodanie głównego komunikatora pomiędzy topelementami do topelementów
*)
METHOD LinkMassangerToaddedTopElements : BOOL
VAR_INPUT
	itfMachineControl	: B_MachineControl.ITF_MCMachineControlConfigure;
END_VAR
END_METHOD

(*			
	RafalOS
	Rafał Osajda		14.11.2025		TC 4024.66
	Podpięcie przyciskow zmiany trybu i stanu
*)
METHOD LinkRequestButtonChange : BOOL
VAR_INPUT
	itfMachineControl	: B_MachineControl.ITF_MCMachineControlConfigure;
END_VAR
END_METHOD

(*			
	RafalOS
	Rafał Osajda		13.11.2025		TC 4024.66
	Podłączenie wsyzstkich zmiennych pochodzących od Programu safety 
*)
METHOD LinkSafetyToaddedElements : BOOL
VAR_INPUT
	itfMachineControl	: B_MachineControl.ITF_MCMachineControlConfigure;
END_VAR
END_METHOD

(*			
	RafalOS
	Rafał Osajda		13.11.2025		TC 4024.66
	Nadanie unikalnych kodów elementom w systemie
*)
METHOD SetCodeToAddedElements : BOOL
VAR_INPUT
	itfMachineControl	: B_MachineControl.ITF_MCMachineControlConfigure;
END_VAR
END_METHOD

(*			
	RafalOS
	Rafał Osajda		13.11.2025		TC 4024.66
	Uruchomienie lub wyłączenie obsługi HMI jak jest false fb obsługi nie jest dodawane do MachineControl
*)
METHOD SetEnableHMIService : BOOL
VAR_INPUT
	itfMachineControl	: B_MachineControl.ITF_MCMachineControlConfigure;
END_VAR
END_METHOD

(*			
	RafalOS
	Rafał Osajda		13.11.2025		TC 4024.66
	Nadaje unikalne ID zgłoszeniom dodanym do elementów w sesyemie
*)
METHOD SetIDEventsToAddedElements : BOOL
VAR_INPUT
	itfMachineControl	: B_MachineControl.ITF_MCMachineControlConfigure;
END_VAR
END_METHOD

(*			
	RafalOS
	Rafał Osajda		13.11.2025		TC 4024.66
	Dodanie wszystkim elementom w systemie unikalnego ID
*)
METHOD SetIDToAddedElements : BOOL
VAR_INPUT
	itfMachineControl	: B_MachineControl.ITF_MCMachineControlConfigure;
END_VAR
END_METHOD

(*			
	RafalOS
	Rafał Osajda		14.11.2025		TC 4024.66
	ustawienie trybu poczatkowego
*)
METHOD SetStartMode : BOOL
VAR_INPUT
	itfMachineControl	: B_MachineControl.ITF_MCMachineControlConfigure;
END_VAR
END_METHOD

END_FUNCTION_BLOCK

// ---- POUs/02_HMIConfiguration/FB_HMIConfiguration.TcPOU
(*			
	RafalOS
	Rafał Osajda		10.11.2025		TC 4024.66
	Główny blok konfigurujący HMI
*)
FUNCTION_BLOCK FB_HMIConfiguration EXTENDS FB_Base IMPLEMENTS ITF_HMIConfiguration
VAR
END_VAR

(*			
	RafalOS
	Rafał Osajda		07.12.2025		TC 4024.66
	Dodawanie elementów do systemmu wyświetlania
*)
METHOD AddElement
VAR_INPUT
	itfHMIManager	: ITF_HMIManagerConfigure;
END_VAR
itfHMIManager.AddElementFromConfiguration (
	fbTopElementHMI := GVL_TE1.fbTopElement1HMI
);

itfHMIManager.AddElementFromConfiguration (
	fbTopElementHMI := GVL_TE2.fbTopElement2HMI
);
END_METHOD

(*			
	RafalOS
	Rafał Osajda		20.11.2025		TC 4024.66
	Dodawanie rozszerzonego wyświetlania danych inna prezenacja danych niż domyślna lista
*)
METHOD AddExtendedDisplayToPrepScrModule : BOOL
VAR_INPUT
	itfHMIManager	: B_HMI_Manager.ITF_HMIManagerConfigure;
END_VAR
END_METHOD

(*			
	RafalOS
	Rafał Osajda		19.11.2025		TC 4024.66
	Dodanie połączenia do MachineControl
*)
METHOD AddMachineControlConnector : BOOL
VAR_INPUT
	itfHMIManager	: B_HMI_Manager.ITF_HMIManagerConfigure;
END_VAR
END_METHOD

(*			
	RafalOS
	Rafał Osajda		14.11.2025		TC 4024.66
	Dodanie do systemu menu głównego 
*)
METHOD AddMainMenu : BOOL
VAR_INPUT
	itfHMIManager	: B_HMI_Manager.ITF_HMIManagerConfigure;
END_VAR
END_METHOD

(*			
	RafalOS
	Rafał Osajda		19.11.2025		TC 4024.66
	Dodanie modułów do przygotowywania stron do wyświetlenia
*)
METHOD AddPrepareScreenModule : BOOL
VAR_INPUT
	itfHMIManager	: B_HMI_Manager.ITF_HMIManagerConfigure;
END_VAR
END_METHOD

(*			
	RafalOS
	Rafał Osajda		26.11.2025		TC 4024.66
	Podłaczenie modułu receptur
*)
METHOD AddRecipeModule : BOOL
VAR_INPUT
	itfHMIManager	: B_HMI_Manager.ITF_HMIManagerConfigure;
END_VAR
END_METHOD

(*			
	RafalOS
	Rafał Osajda		18.11.2025		TC 4024.66
	Podłączenie głównej struktury danych dla domyślnych elementów 
*)
METHOD LinkCommonStructureData : BOOL
VAR_INPUT
	itfHMIManager	: B_HMI_Manager.ITF_HMIManagerConfigure;
END_VAR
END_METHOD

METHOD LinkHMIManagerData : BOOL
VAR_INPUT
	itfHMIManager	: B_HMI_Manager.ITF_HMIManagerConfigure;
END_VAR
END_METHOD

METHOD LinkMachineData : BOOL
VAR_INPUT
	itfHMIManager	: B_HMI_Manager.ITF_HMIManagerConfigure;
END_VAR
GVL_TE1.fbTopElement1HMI.LinkTopElementData (stData := GVL_TE1.stTopElemenent1);
GVL_TE2.fbTopElement2HMI.LinkTopElementData (stData := GVL_TE2.stTopElemenent2);
END_METHOD

(*			
	RafalOS
	Rafał Osajda		13.11.2025		TC 4024.66
	Podłączenie wsyzstkich zmiennych pochodzących od Programu safety 
*)
METHOD LinkSafetyToaddedElements : BOOL
VAR_INPUT
	itfHMIManager	: B_HMI_Manager.ITF_HMIManagerConfigure;
END_VAR
END_METHOD

(*			
	RafalOS
	Rafał Osajda		18.11.2025		TC 4024.66
	Ustawia przycisk na aktywny  - pierwsze okno w wyświetlaniu wizualizacji
*)
METHOD SetButtonActive : BOOL
VAR_INPUT
	itfHMIManager	: B_HMI_Manager.ITF_HMIManagerConfigure;
END_VAR
END_METHOD

(*			
	RafalOS
	Rafał Osajda		18.11.2025		TC 4024.66
	Ustawia przyciski na wlaczone lub wylaczone - możliwośc naciśnięcia
*)
METHOD SetButtonsEnabled : BOOL
VAR_INPUT
	itfHMIManager	: B_HMI_Manager.ITF_HMIManagerConfigure;
END_VAR

VAR
	iI					: INT;
	iNumberofButtons	: INT;
END_VAR
END_METHOD

(*			
	RafalOS
	Rafał Osajda		18.11.2025		TC 4024.66
	Ustawia przyciski na widoczne lub nie widoczne
*)
METHOD SetButtonsVisible : BOOL
VAR_INPUT
	itfHMIManager	: B_HMI_Manager.ITF_HMIManagerConfigure;
END_VAR
VAR
	iI					: INT;
	iNumberofButtons	: INT;
END_VAR
itfHMIManager.SetButtonsVisibleFromConfiguration (iNumber := 5, bValue := FALSE);
END_METHOD

END_FUNCTION_BLOCK

// ---- POUs/03_CreatingTemplateRecipe/FB_MachineTemplate1.TcPOU
FUNCTION_BLOCK FB_MachineTemplate1 EXTENDS FB_Base IMPLEMENTS ITF_BaseCreateTemplateOfRecipe
VAR
END_VAR

METHOD CreateTamplateOfRecipe : BOOL
VAR_INPUT
	(*interfejs do obsługi receptur*)
	itfRecipe	: B_Base.ITF_BaseCreatingTemplateMethod;
END_VAR
VAR
	sttmpSkladnik			: ST_BaseDescriptor;
	uiNumberOfTeplates		: UINT;
END_VAR
(*	Metody tworzące szablon receptury 
	- dodanie nazwy i utworzenie szablonu 
	- dodawanie składników
*)

//	utworzenie szablonu z podaną nazwą
THIS^.SetText (eLocation := E_BaseLocation.pl, wsDescription := "Nazwa szablonu PL");
THIS^.SetText (eLocation := E_BaseLocation.en, wsDescription := "Nazwa szablonu EN");
THIS^.SetText (eLocation := E_BaseLocation.de, wsDescription := "Nazwa szablonu DE");
itfRecipe.AddTemplate (stTexts	:= THIS^.GetTexts ());
uiNumberOfTeplates	:= itfRecipe.GetNumberOfTemplate ();

THIS^.SetTextIn (stIN := sttmpSkladnik, eLocation := E_BaseLocation.pl, wsDescription := "Nazwa skladnika 1 PL");
THIS^.SetTextIn (stIN := sttmpSkladnik, eLocation := E_BaseLocation.en, wsDescription := "Nazwa skladnika 1 EN");
THIS^.SetTextIn (stIN := sttmpSkladnik, eLocation := E_BaseLocation.de, wsDescription := "Nazwa skladnika 1 DE");
THIS^.SetMaxIn (stIN := sttmpSkladnik, rMax := 10000);
THIS^.SetMinIn (stIN := sttmpSkladnik, rMin := 1);
THIS^.SetValueIn (stIN := sttmpSkladnik, rValue := 1111);
THIS^.SetDefaultValueIn (stIN := sttmpSkladnik, rDefaultValue := 1111);
THIS^.SetUnitIn (stIN := sttmpSkladnik, sUnit := 'mm');
itfRecipe.AddIngredientToTemplate (uiNumber := uiNumberOfTeplates, stIngredient := sttmpSkladnik);

THIS^.SetTextIn (stIN := sttmpSkladnik, eLocation := E_BaseLocation.pl, wsDescription := "Nazwa skladnika 2 PL");
THIS^.SetTextIn (stIN := sttmpSkladnik, eLocation := E_BaseLocation.en, wsDescription := "Nazwa skladnika 2 EN");
THIS^.SetTextIn (stIN := sttmpSkladnik, eLocation := E_BaseLocation.de, wsDescription := "Nazwa skladnika 2 DE");
THIS^.SetMaxIn (stIN := sttmpSkladnik, rMax := 10000);
THIS^.SetMinIn (stIN := sttmpSkladnik, rMin := 1);
THIS^.SetValueIn (stIN := sttmpSkladnik, rValue := 1112);
THIS^.SetDefaultValueIn (stIN := sttmpSkladnik, rDefaultValue := 1112);
THIS^.SetUnitIn (stIN := sttmpSkladnik, sUnit := 'mm/s');
itfRecipe.AddIngredientToTemplate (uiNumber := uiNumberOfTeplates, stIngredient := sttmpSkladnik);

THIS^.SetTextIn (stIN := sttmpSkladnik, eLocation := E_BaseLocation.pl, wsDescription := "Nazwa skladnika 3 PL");
THIS^.SetTextIn (stIN := sttmpSkladnik, eLocation := E_BaseLocation.en, wsDescription := "Nazwa skladnika 3 EN");
THIS^.SetTextIn (stIN := sttmpSkladnik, eLocation := E_BaseLocation.de, wsDescription := "Nazwa skladnika 3 DE");
THIS^.SetMaxIn (stIN := sttmpSkladnik, rMax := 10000);
THIS^.SetMinIn (stIN := sttmpSkladnik, rMin := 1);
THIS^.SetValueIn (stIN := sttmpSkladnik, rValue := 1113);
THIS^.SetDefaultValueIn (stIN := sttmpSkladnik, rDefaultValue := 1113);
THIS^.SetUnitIn (stIN := sttmpSkladnik, sUnit := 'ms');
itfRecipe.AddIngredientToTemplate (uiNumber := uiNumberOfTeplates, stIngredient := sttmpSkladnik);
END_METHOD

END_FUNCTION_BLOCK

// ---- POUs/03_CreatingTemplateRecipe/FB_MachineTemplate2.TcPOU
FUNCTION_BLOCK FB_MachineTemplate2 EXTENDS FB_Base IMPLEMENTS ITF_BaseCreateTemplateOfRecipe
VAR
END_VAR

METHOD CreateTamplateOfRecipe : BOOL
VAR_INPUT
	(*interfejs do obsługi receptur*)
	itfRecipe	: B_Base.ITF_BaseCreatingTemplateMethod;
END_VAR
VAR
	sttmpSkladnik			: ST_BaseDescriptor;
	uiNumberOfTeplates		: UINT;
END_VAR
(*	Metody tworzące szablon receptury 
	- dodanie nazwy i utworzenie szablonu 
	- dodawanie składników
*)
THIS^.SetText (eLocation := E_BaseLocation.pl, wsDescription := "Nazwa szablonu 2 PL");
THIS^.SetText (eLocation := E_BaseLocation.en, wsDescription := "Nazwa szablonu 2 EN");
THIS^.SetText (eLocation := E_BaseLocation.de, wsDescription := "Nazwa szablonu 2 DE");
itfRecipe.AddTemplate (stTexts	:= THIS^.GetTexts ());
uiNumberOfTeplates	:= itfRecipe.GetNumberOfTemplate ();

THIS^.SetTextIn (stIN := sttmpSkladnik, eLocation := E_BaseLocation.pl, wsDescription := "Nazwa skladnika 1 PL");
THIS^.SetTextIn (stIN := sttmpSkladnik, eLocation := E_BaseLocation.en, wsDescription := "Nazwa skladnika 1 EN");
THIS^.SetTextIn (stIN := sttmpSkladnik, eLocation := E_BaseLocation.de, wsDescription := "Nazwa skladnika 1 DE");
THIS^.SetMaxIn (stIN := sttmpSkladnik, rMax := 10000);
THIS^.SetMinIn (stIN := sttmpSkladnik, rMin := 1);
THIS^.SetValueIn (stIN := sttmpSkladnik, rValue := 1111);
THIS^.SetDefaultValueIn (stIN := sttmpSkladnik, rDefaultValue := 1111);
THIS^.SetUnitIn (stIN := sttmpSkladnik, sUnit := 'mm');
itfRecipe.AddIngredientToTemplate (uiNumber := uiNumberOfTeplates, stIngredient := sttmpSkladnik);
END_METHOD

END_FUNCTION_BLOCK

// ---- POUs/03_CreatingTemplateRecipe/FB_MachineTemplate3.TcPOU
FUNCTION_BLOCK FB_MachineTemplate3 EXTENDS FB_Base IMPLEMENTS ITF_BaseCreateTemplateOfRecipe
VAR
END_VAR

METHOD CreateTamplateOfRecipe : BOOL
VAR_INPUT
	(*interfejs do obsługi receptur*)
	itfRecipe	: B_Base.ITF_BaseCreatingTemplateMethod;
END_VAR
VAR
	sttmpSkladnik			: ST_BaseDescriptor;
	uiNumberOfTeplates		: UINT;
	iI						: INT;
	wstmpDescription		: WSTRING;
END_VAR
(*	Metody tworzące szablon receptury 
	- dodanie nazwy i utworzenie szablonu 
	- dodawanie składników
*)
THIS^.SetText (eLocation := E_BaseLocation.pl, wsDescription := "Nazwa szablonu 3 PL");
THIS^.SetText (eLocation := E_BaseLocation.en, wsDescription := "Nazwa szablonu 3 EN");
THIS^.SetText (eLocation := E_BaseLocation.de, wsDescription := "Nazwa szablonu 3 DE");
itfRecipe.AddTemplate (stTexts	:= THIS^.GetTexts ());
uiNumberOfTeplates	:= itfRecipe.GetNumberOfTemplate ();

FOR iI := 1 TO 115 DO
	THIS^.SetTextIn (stIN := sttmpSkladnik, eLocation := E_BaseLocation.pl, wsDescription := wconcat ("Nazwa składnika PL ", TO_WSTRING (iI)));
	THIS^.SetTextIn (stIN := sttmpSkladnik, eLocation := E_BaseLocation.en, wsDescription := wconcat ("Nazwa składnika PL ", TO_WSTRING (iI)));
	THIS^.SetTextIn (stIN := sttmpSkladnik, eLocation := E_BaseLocation.de, wsDescription := wconcat ("Nazwa składnika PL ", TO_WSTRING (iI)));
	THIS^.SetMaxIn (stIN := sttmpSkladnik, rMax := 10000+iI);
	THIS^.SetMinIn (stIN := sttmpSkladnik, rMin := 1);
	THIS^.SetValueIn (stIN := sttmpSkladnik, rValue := iI);
	THIS^.SetDefaultValueIn (stIN := sttmpSkladnik, rDefaultValue := iI);
	THIS^.SetUnitIn (stIN := sttmpSkladnik, sUnit := 'mm');
	itfRecipe.AddIngredientToTemplate (uiNumber := uiNumberOfTeplates, stIngredient := sttmpSkladnik);
END_FOR
END_METHOD

END_FUNCTION_BLOCK

// ---- POUs/04_TopElement1/1C_B/FB_Component_TE1.TcPOU
FUNCTION_BLOCK FB_Component_TE1 EXTENDS FB_BaseComponent IMPLEMENTS ITF_Component_TE1, ITF_Component_TE1_HMI_Init
VAR
END_VAR

METHOD testMethod : BOOL
VAR_INPUT
END_VAR
END_METHOD

END_FUNCTION_BLOCK

// ---- POUs/04_TopElement1/2CE_B/FB_ControlE_TE1.TcPOU
FUNCTION_BLOCK FB_ControlE_TE1 EXTENDS FB_BaseControlElement IMPLEMENTS ITF_ControlE_TE1, ITF_ControlE_TE1_HMI_Init
VAR
	itfC1				: ITF_Component_TE1;
	itfC2				: ITF_Component_TE1;
	itfC3				: ITF_Component_TE1;
	itfC4				: ITF_Component_TE1;
	
END_VAR

METHOD FB_init : BOOL
VAR_INPUT
	bInitRetains : BOOL; // if TRUE, the retain variables are initialized (warm start / cold start)
	bInCopyCode : BOOL;  // if TRUE, the instance afterwards gets moved into the copy code (online change)
	itfC1				: ITF_Component_TE1;
	itfC2				: ITF_Component_TE1;
	itfC3				: ITF_Component_TE1;
	itfC4				: ITF_Component_TE1;
END_VAR
THIS^.itfC1 := itfC1;
THIS^.SetText (eLocation := E_BaseLocation.pl, wsDescription := "Komponent 1 EC");
THIS^.SetText (eLocation := E_BaseLocation.en, wsDescription := "Komponent 1 EC");
THIS^.SetText (eLocation := E_BaseLocation.de, wsDescription := "Komponent 1 EC");
itfC1.SetName (stName := THIS^.GetTexts ());
THIS^.AddComponent (itfComponent := itfC1);

THIS^.itfC2 := itfC2;
THIS^.SetText (eLocation := E_BaseLocation.pl, wsDescription := "Komponent 2 EC");
THIS^.SetText (eLocation := E_BaseLocation.en, wsDescription := "Komponent 2 EC");
THIS^.SetText (eLocation := E_BaseLocation.de, wsDescription := "Komponent 2 EC");
itfC2.SetName (stName := THIS^.GetTexts ());
THIS^.AddComponent (itfComponent := itfC2);

THIS^.itfC3 := itfC3;
THIS^.SetText (eLocation := E_BaseLocation.pl, wsDescription := "Komponent 3 EC");
THIS^.SetText (eLocation := E_BaseLocation.en, wsDescription := "Komponent 3 EC");
THIS^.SetText (eLocation := E_BaseLocation.de, wsDescription := "Komponent 3 EC");
itfC3.SetName (stName := THIS^.GetTexts ());
THIS^.AddComponent (itfComponent := itfC3);

THIS^.itfC4 := itfC4;
THIS^.SetText (eLocation := E_BaseLocation.pl, wsDescription := "Komponent 4 EC");
THIS^.SetText (eLocation := E_BaseLocation.en, wsDescription := "Komponent 4 EC");
THIS^.SetText (eLocation := E_BaseLocation.de, wsDescription := "Komponent 4 EC");
itfC4.SetName (stName := THIS^.GetTexts ());
THIS^.AddComponent (itfComponent := itfC4);
END_METHOD

METHOD testMethodCE : BOOL
VAR_INPUT
END_VAR
END_METHOD

END_FUNCTION_BLOCK

// ---- POUs/04_TopElement1/3GE_B/FB_GroupE_TE1.TcPOU
FUNCTION_BLOCK FB_GroupE_TE1 EXTENDS FB_BaseGroupElement IMPLEMENTS ITF_GroupE_TE1, ITF_GroupE_TE1_HMI_Init
VAR
	itfCE1				: ITF_ControlE_TE1;
	itfCE2				: ITF_ControlE_TE1;

	itfC1				: ITF_Component_TE1;
	itfC2				: ITF_Component_TE1;
	itfC3				: ITF_Component_TE1;
	itfC4				: ITF_Component_TE1;
	
END_VAR

METHOD FB_init : BOOL
VAR_INPUT
	bInitRetains : BOOL; // if TRUE, the retain variables are initialized (warm start / cold start)
	bInCopyCode : BOOL;  // if TRUE, the instance afterwards gets moved into the copy code (online change)
	itfCE1				: ITF_ControlE_TE1;
	itfCE2				: ITF_ControlE_TE1;
	itfC1				: ITF_Component_TE1;
	itfC2				: ITF_Component_TE1;
	itfC3				: ITF_Component_TE1;
	itfC4				: ITF_Component_TE1;
END_VAR
THIS^.itfCE1 := itfCE1;
THIS^.SetText (eLocation := E_BaseLocation.pl, wsDescription := "Element 1 EC");
THIS^.SetText (eLocation := E_BaseLocation.en, wsDescription := "Element 1 EC");
THIS^.SetText (eLocation := E_BaseLocation.de, wsDescription := "Element 1 EC");
itfCE1.SetName (stName := THIS^.GetTexts ());
THIS^.AddControlElement (itfControlElement := itfCE1);

THIS^.itfCE2 := itfCE2;
THIS^.SetText (eLocation := E_BaseLocation.pl, wsDescription := "Element 2 EC");
THIS^.SetText (eLocation := E_BaseLocation.en, wsDescription := "Element 2 EC");
THIS^.SetText (eLocation := E_BaseLocation.de, wsDescription := "Element 2 EC");
itfCE2.SetName (stName := THIS^.GetTexts ());
THIS^.AddControlElement (itfControlElement := itfCE2);

THIS^.itfC1 := itfC1;
THIS^.SetText (eLocation := E_BaseLocation.pl, wsDescription := "Komponent 1 EC");
THIS^.SetText (eLocation := E_BaseLocation.en, wsDescription := "Komponent 1 EC");
THIS^.SetText (eLocation := E_BaseLocation.de, wsDescription := "Komponent 1 EC");
itfC1.SetName (stName := THIS^.GetTexts ());
THIS^.AddComponent (itfComponent := itfC1);

THIS^.itfC2 := itfC2;
THIS^.SetText (eLocation := E_BaseLocation.pl, wsDescription := "Komponent 2 EC");
THIS^.SetText (eLocation := E_BaseLocation.en, wsDescription := "Komponent 2 EC");
THIS^.SetText (eLocation := E_BaseLocation.de, wsDescription := "Komponent 2 EC");
itfC2.SetName (stName := THIS^.GetTexts ());
THIS^.AddComponent (itfComponent := itfC2);

THIS^.itfC3 := itfC3;
THIS^.SetText (eLocation := E_BaseLocation.pl, wsDescription := "Komponent 3 EC");
THIS^.SetText (eLocation := E_BaseLocation.en, wsDescription := "Komponent 3 EC");
THIS^.SetText (eLocation := E_BaseLocation.de, wsDescription := "Komponent 3 EC");
itfC3.SetName (stName := THIS^.GetTexts ());
THIS^.AddComponent (itfComponent := itfC3);

THIS^.itfC4 := itfC4;
THIS^.SetText (eLocation := E_BaseLocation.pl, wsDescription := "Komponent 4 EC");
THIS^.SetText (eLocation := E_BaseLocation.en, wsDescription := "Komponent 4 EC");
THIS^.SetText (eLocation := E_BaseLocation.de, wsDescription := "Komponent 4 EC");
itfC4.SetName (stName := THIS^.GetTexts ());
THIS^.AddComponent (itfComponent := itfC4);
END_METHOD

METHOD testMethodGE : BOOL
VAR_INPUT
END_VAR
END_METHOD

END_FUNCTION_BLOCK

// ---- POUs/04_TopElement1/9TE_B/FB_TopElement1.TcPOU
FUNCTION_BLOCK FB_TopElement1 EXTENDS FB_BaseTopElement IMPLEMENTS ITF_TopElement1, ITF_TopElement1_HMI_Init
VAR
	itfGE1				: ITF_GroupE_TE1;

	itfCE1				: ITF_ControlE_TE1;
	itfCE2				: ITF_ControlE_TE1;

	itfC1				: ITF_Component_TE1;
	itfC2				: ITF_Component_TE1;
	itfC3				: ITF_Component_TE1;
END_VAR

METHOD FB_init : BOOL
VAR_INPUT
	bInitRetains : BOOL; // if TRUE, the retain variables are initialized (warm start / cold start)
	bInCopyCode : BOOL;  // if TRUE, the instance afterwards gets moved into the copy code (online change)
	itfGE1				: ITF_GroupE_TE1;
	itfCE1				: ITF_ControlE_TE1;
	itfCE2				: ITF_ControlE_TE1;
	itfC1				: ITF_Component_TE1;
	itfC2				: ITF_Component_TE1;
	itfC3				: ITF_Component_TE1;
END_VAR
THIS^.itfGE1 := itfGE1;
THIS^.SetText (eLocation := E_BaseLocation.pl, wsDescription := "Element złożony 1");
THIS^.SetText (eLocation := E_BaseLocation.en, wsDescription := "Element złożony 1");
THIS^.SetText (eLocation := E_BaseLocation.de, wsDescription := "Element złożony 1");
itfGE1.SetName (stName := THIS^.GetTexts ());
THIS^.AddControlElement (itfControlElement := itfGE1);

THIS^.itfCE1 := itfCE1;
THIS^.SetText (eLocation := E_BaseLocation.pl, wsDescription := "Element wykonawczy 1");
THIS^.SetText (eLocation := E_BaseLocation.en, wsDescription := "Element wykonawczy 1");
THIS^.SetText (eLocation := E_BaseLocation.de, wsDescription := "Element wykonawczy 1");
itfCE1.SetName (stName := THIS^.GetTexts ());
THIS^.AddControlElement (itfControlElement := itfCE1);

THIS^.itfCE2 := itfCE2;
THIS^.SetText (eLocation := E_BaseLocation.pl, wsDescription := "Element wykonawczy 2");
THIS^.SetText (eLocation := E_BaseLocation.en, wsDescription := "Element wykonawczy 2");
THIS^.SetText (eLocation := E_BaseLocation.de, wsDescription := "Element wykonawczy 2");
itfCE2.SetName (stName := THIS^.GetTexts ());
THIS^.AddControlElement (itfControlElement := itfCE2);


THIS^.itfC1 := itfC1;
THIS^.SetText (eLocation := E_BaseLocation.pl, wsDescription := "Komponent 1");
THIS^.SetText (eLocation := E_BaseLocation.en, wsDescription := "Komponent 1");
THIS^.SetText (eLocation := E_BaseLocation.de, wsDescription := "Komponent 1");
itfC1.SetName (stName := THIS^.GetTexts ());
THIS^.AddComponent (itfComponent := itfC1);

THIS^.itfC2 := itfC2;
THIS^.SetText (eLocation := E_BaseLocation.pl, wsDescription := "Komponent 2");
THIS^.SetText (eLocation := E_BaseLocation.en, wsDescription := "Komponent 2");
THIS^.SetText (eLocation := E_BaseLocation.de, wsDescription := "Komponent 2");
itfC2.SetName (stName := THIS^.GetTexts ());
THIS^.AddComponent (itfComponent := itfC2);

THIS^.itfC3 := itfC3;
THIS^.SetText (eLocation := E_BaseLocation.pl, wsDescription := "Komponent 3");
THIS^.SetText (eLocation := E_BaseLocation.en, wsDescription := "Komponent 3");
THIS^.SetText (eLocation := E_BaseLocation.de, wsDescription := "Komponent 3");
itfC3.SetName (stName := THIS^.GetTexts ());
THIS^.AddComponent (itfComponent := itfC3);
END_METHOD

END_FUNCTION_BLOCK

// ---- POUs/04_TopElement1/1C_B_HMI/FB_Component_TE1_HMI.TcPOU
FUNCTION_BLOCK FB_Component_TE1_HMI EXTENDS FB_BaseComponent_HMI IMPLEMENTS ITF_Component_TE1_HMI
VAR
	itfComponent_TE1Connector		: ITF_Component_TE1_HMI_Connector;
	refstComponent_TE1Data			: REFERENCE TO ST_Component_TE1_HMI;

	
END_VAR

METHOD FB_init : BOOL
VAR_INPUT
	bInitRetains : BOOL; // if TRUE, the retain variables are initialized (warm start / cold start)
	bInCopyCode : BOOL;  // if TRUE, the instance afterwards gets moved into the copy code (online change)
	itfBaseLoggerConnector				: ITF_BaseLogger_HMI_Connector;	//bezpośredni łącznik do logera
	itfComponent_TE1Connector			: ITF_Component_TE1_HMI_Init;
END_VAR
//Przypisanie do elementu który własnie stworzyliśmy
THIS^.itfComponent_TE1Connector			:= itfComponent_TE1Connector;
//Przypisanie do elementów z biblioteki
THIS^.itfBaseLoggerElementConnector		:= itfComponent_TE1Connector;
THIS^.itfBaseComponentConnector			:= itfComponent_TE1Connector;

//
THIS^.itfBaseLoggerConnector			:= itfBaseLoggerConnector;

IF (THIS^.itfComponent_TE1Connector <> 0 AND
	THIS^.itfBaseLoggerElementConnector <> 0 AND
	THIS^.itfBaseComponentConnector	<> 0 AND
	THIS^.itfBaseLoggerConnector <> 0) THEN
	THIS^.bIsInit						:= TRUE;
END_IF
END_METHOD

METHOD LinkComponentData : BOOL
VAR_INPUT
	stData				: REFERENCE TO ST_Component_TE1_HMI_Link;
END_VAR
THIS^.refstComponent_TE1Data REF= stData.stComponent_TE1;

THIS^.refstBaseLoggerElementDataHMI REF= stData.stBaseLoggerElement;
THIS^.refstBaseComponentDataHMI REF= stData.stBaseComponent;



THIS^.CreateLinkToEventsMemory ();

IF (__ISVALIDREF (THIS^.refstComponent_TE1Data) AND this^.IsLinkedReferences ()) THEN
	THIS^.bIsValidData		:= TRUE;
	LinkComponentData		:= TRUE;
END_IF
END_METHOD

END_FUNCTION_BLOCK

// ---- POUs/04_TopElement1/2CE_B_HMI/FB_ControlE_TE1_HMI.TcPOU
FUNCTION_BLOCK FB_ControlE_TE1_HMI EXTENDS FB_BaseControlElement_HMI IMPLEMENTS ITF_ControlE_TE1_HMI
VAR
	itfControlE_TE1Connector		: ITF_ControlE_TE1_HMI_Connector;
	refstControlE_TE1Data			: REFERENCE TO ST_ControlE_TE1_HMI;

	itfC1				: ITF_Component_TE1_HMI;
	itfC2				: ITF_Component_TE1_HMI;
	itfC3				: ITF_Component_TE1_HMI;
	itfC4				: ITF_Component_TE1_HMI;
	
END_VAR

METHOD FB_init : BOOL
VAR_INPUT
	bInitRetains : BOOL; // if TRUE, the retain variables are initialized (warm start / cold start)
	bInCopyCode : BOOL;  // if TRUE, the instance afterwards gets moved into the copy code (online change)
	itfBaseLoggerConnector				: ITF_BaseLogger_HMI_Connector;	//bezpośredni łącznik do logera
	itfControlE_TE1Connector			: ITF_ControlE_TE1_HMI_Connector;
	itfC1								: ITF_Component_TE1_HMI;
	itfC2								: ITF_Component_TE1_HMI;
	itfC3								: ITF_Component_TE1_HMI;
	itfC4								: ITF_Component_TE1_HMI;
END_VAR
//Przypisanie do elementu który własnie stworzyliśmy
THIS^.itfControlE_TE1Connector := itfControlE_TE1Connector;
//Przypisanie do elementów z biblioteki
THIS^.itfBaseLoggerElementConnector := itfControlE_TE1Connector;
THIS^.itfBaseComponentConnector := itfControlE_TE1Connector;
THIS^.itfBaseControlElementConnector := itfControlE_TE1Connector;

THIS^.AddComponent (itfComponentHMI := itfC1);
THIS^.itfC1 := itfC1;
THIS^.AddComponent (itfComponentHMI := itfC2);
THIS^.itfC2 := itfC2;
THIS^.AddComponent (itfComponentHMI := itfC3);
THIS^.itfC3 := itfC3;
THIS^.AddComponent (itfComponentHMI := itfC4);
THIS^.itfC4 := itfC4;


//
THIS^.itfBaseLoggerConnector			:= itfBaseLoggerConnector;

IF (THIS^.itfControlE_TE1Connector <> 0 AND
	THIS^.itfBaseLoggerElementConnector <> 0 AND
	THIS^.itfBaseComponentConnector	<> 0 AND
	THIS^.itfBaseControlElementConnector <> 0 AND
	THIS^.itfBaseLoggerConnector <> 0) THEN
	THIS^.bIsInit						:= TRUE;
END_IF
END_METHOD

METHOD LinkControlEData : BOOL
VAR_INPUT
	stData				: REFERENCE TO ST_ControlE_TE1_HMI_Link;
END_VAR
THIS^.refstControlE_TE1Data REF= stData.stControlE_TE1;

THIS^.refstBaseLoggerElementDataHMI REF= stData.stBaseLoggerElement;
THIS^.refstBaseComponentDataHMI REF= stData.stBaseComponent;
THIS^.refstBaseControlElementDataHMI REF= stData.stBaseControlElement;

THIS^.itfC1.LinkComponentData (stData := stData.stComponetE1_TE1);
THIS^.itfC2.LinkComponentData (stData := stData.stComponetE2_TE1);
THIS^.itfC3.LinkComponentData (stData := stData.stComponetE3_TE1);
THIS^.itfC4.LinkComponentData (stData := stData.stComponetE4_TE1);


THIS^.CreateLinkToEventsMemory ();

IF (__ISVALIDREF (THIS^.refstControlE_TE1Data) AND THIS^.IsLinkedReferences ()) THEN
	THIS^.bIsValidData		:= TRUE;
	LinkControlEData		:= TRUE;
END_IF
END_METHOD

END_FUNCTION_BLOCK

// ---- POUs/04_TopElement1/3GE_B_HMI/FB_GroupE_TE1_HMI.TcPOU
FUNCTION_BLOCK FB_GroupE_TE1_HMI EXTENDS FB_BaseGroupElement_HMI IMPLEMENTS ITF_GroupE_TE1_HMI
VAR
	itfGroupE_TE1Connector		: ITF_GroupE_TE1_HMI_Connector;
	refstGroupE_TE1Data			: REFERENCE TO ST_GroupE_TE1_HMI;
	
	itfCE1				: ITF_ControlE_TE1_HMI;
	itfCE2				: ITF_ControlE_TE1_HMI;

	itfC1				: ITF_Component_TE1_HMI;
	itfC2				: ITF_Component_TE1_HMI;
	itfC3				: ITF_Component_TE1_HMI;
	itfC4				: ITF_Component_TE1_HMI;
	
END_VAR

METHOD FB_init : BOOL
VAR_INPUT
	bInitRetains : BOOL; // if TRUE, the retain variables are initialized (warm start / cold start)
	bInCopyCode : BOOL;  // if TRUE, the instance afterwards gets moved into the copy code (online change)
	itfBaseLoggerConnector			: ITF_BaseLogger_HMI_Connector;	//bezpośredni łącznik do logera
	itfGroupE_TE1Connector			: ITF_GroupE_TE1_HMI_Connector;
	itfCE1							: ITF_ControlE_TE1_HMI;
	itfCE2							: ITF_ControlE_TE1_HMI;
	itfC1								: ITF_Component_TE1_HMI;
	itfC2								: ITF_Component_TE1_HMI;
	itfC3								: ITF_Component_TE1_HMI;
	itfC4								: ITF_Component_TE1_HMI;
END_VAR
//Przypisanie do elementu który własnie stworzyliśmy
THIS^.itfGroupE_TE1Connector := itfGroupE_TE1Connector;
//Przypisanie do elementów z biblioteki
THIS^.itfBaseLoggerElementConnector := itfGroupE_TE1Connector;
THIS^.itfBaseComponentConnector := itfGroupE_TE1Connector;
THIS^.itfBaseControlElementConnector := itfGroupE_TE1Connector;
THIS^.itfBaseGroupElementConnector := itfGroupE_TE1Connector;

THIS^.AddControlElement (itfControlElementHMI := itfCE1);
THIS^.itfCE1 := itfCE1;
THIS^.AddControlElement (itfControlElementHMI := itfCE2);
THIS^.itfCE2 := itfCE2;

THIS^.AddComponent (itfComponentHMI := itfC1);
THIS^.itfC1 := itfC1;
THIS^.AddComponent (itfComponentHMI := itfC2);
THIS^.itfC2 := itfC2;
THIS^.AddComponent (itfComponentHMI := itfC3);
THIS^.itfC3 := itfC3;
THIS^.AddComponent (itfComponentHMI := itfC4);
THIS^.itfC4 := itfC4;


//
THIS^.itfBaseLoggerConnector			:= itfBaseLoggerConnector;

IF (THIS^.itfGroupE_TE1Connector <> 0 AND
	THIS^.itfBaseLoggerElementConnector <> 0 AND
	THIS^.itfBaseComponentConnector	<> 0 AND
	THIS^.itfBaseControlElementConnector <> 0 AND
	THIS^.itfBaseGroupElementConnector <> 0 AND
	THIS^.itfBaseLoggerConnector <> 0) THEN
	THIS^.bIsInit						:= TRUE;
END_IF
END_METHOD

METHOD LinkGroupEData : BOOL
VAR_INPUT
	stData				: REFERENCE TO ST_GroupE_TE1_HMI_Link;
END_VAR
THIS^.refstGroupE_TE1Data REF= stData.stGroupE_TE1;

THIS^.refstBaseLoggerElementDataHMI REF= stData.stBaseLoggerElement;
THIS^.refstBaseComponentDataHMI REF= stData.stBaseComponent;
THIS^.refstBaseControlElementDataHMI REF= stData.stBaseControlElement;
THIS^.refstBaseGroupElementDataHMI REF= stData.stBaseGroupElement;

THIS^.itfCE1.LinkControlEData (stData := stData.stControlE1_TE1);
THIS^.itfCE2.LinkControlEData (stData := stData.stControlE2_TE1);

THIS^.itfC1.LinkComponentData (stData := stData.stComponetE1_TE1);
THIS^.itfC2.LinkComponentData (stData := stData.stComponetE2_TE1);
THIS^.itfC3.LinkComponentData (stData := stData.stComponetE3_TE1);
THIS^.itfC4.LinkComponentData (stData := stData.stComponetE4_TE1);


THIS^.CreateLinkToEventsMemory ();

IF (__ISVALIDREF (THIS^.refstGroupE_TE1Data) AND THIS^.IsLinkedReferences ()) THEN
	THIS^.bIsValidData		:= TRUE;
	LinkGroupEData		:= TRUE;
END_IF
END_METHOD

END_FUNCTION_BLOCK

// ---- POUs/04_TopElement1/9TE_B_HMI/FB_TopElement1_HMI.TcPOU
FUNCTION_BLOCK FB_TopElement1_HMI EXTENDS FB_BaseTopElement_HMI IMPLEMENTS ITF_TopElement1_HMI
VAR
	itfTopElementConnector			: ITF_TopElement1_HMI_Connector;
	refstTopElementData				: REFERENCE TO ST_TopElement1_HMI;
	
	itfGE1							: ITF_GroupE_TE1_HMI;
	
	itfCE1							: ITF_ControlE_TE1_HMI;
	itfCE2							: ITF_ControlE_TE1_HMI;
	
	itfC1							: ITF_Component_TE1_HMI;
	itfC2							: ITF_Component_TE1_HMI;
	itfC3							: ITF_Component_TE1_HMI;
END_VAR

METHOD FB_init : BOOL
VAR_INPUT
	bInitRetains : BOOL; // if TRUE, the retain variables are initialized (warm start / cold start)
	bInCopyCode : BOOL;  // if TRUE, the instance afterwards gets moved into the copy code (online change)
	itfBaseLoggerConnector				: ITF_BaseLogger_HMI_Connector;	//bezpośredni łącznik do logera
	itfTopElementConnector				: ITF_TopElement1_HMI_Init;
	itfGE1								: ITF_GroupE_TE1_HMI;
	itfCE1								: ITF_ControlE_TE1_HMI;
	itfCE2								: ITF_ControlE_TE1_HMI;
	itfC1								: ITF_Component_TE1_HMI;
	itfC2								: ITF_Component_TE1_HMI;
	itfC3								: ITF_Component_TE1_HMI;
END_VAR
//Przypisanie do elementu który własnie stworzyliśmy
THIS^.itfTopElementConnector			:= itfTopElementConnector;
//Przypisanie do elementów z biblioteki
THIS^.itfBaseLoggerElementConnector		:= itfTopElementConnector;
THIS^.itfBaseComponentConnector			:= itfTopElementConnector;
THIS^.itfBaseControlElementConnector	:= itfTopElementConnector;
THIS^.itfBaseGroupElementConnector		:= itfTopElementConnector;
THIS^.itfBaseTopElementConnector		:= itfTopElementConnector;
//
THIS^.itfBaseLoggerConnector			:= itfBaseLoggerConnector;

THIS^.AddControlElement (itfControlElementHMI := itfGE1);
THIS^.itfGE1 := itfGE1;

THIS^.AddControlElement (itfControlElementHMI := itfCE1);
THIS^.itfCE1 := itfCE1;

THIS^.AddControlElement (itfControlElementHMI := itfCE2);
THIS^.itfCE2 := itfCE2;

THIS^.AddComponent (itfComponentHMI := itfC1);
THIS^.itfC1 := itfC1;

THIS^.AddComponent (itfComponentHMI := itfC2);
THIS^.itfC2 := itfC2;

THIS^.AddComponent (itfComponentHMI := itfC3);
THIS^.itfC3 := itfC3;

IF (THIS^.itfTopElementConnector <> 0 AND
	THIS^.itfBaseLoggerElementConnector <> 0 AND
	THIS^.itfBaseComponentConnector	<> 0 AND
	THIS^.itfBaseControlElementConnector <> 0 AND
	THIS^.itfBaseGroupElementConnector <> 0 AND
	THIS^.itfBaseTopElementConnector <> 0 AND
	THIS^.itfBaseLoggerConnector <> 0) THEN
	THIS^.bIsInit						:= TRUE;
END_IF
END_METHOD

METHOD LinkTopElementData : BOOL
VAR_INPUT
	stData				: REFERENCE TO ST_TopElement1_HMI_Link;
END_VAR

VAR
	stBaseGroupElem: INT;
END_VAR
THIS^.refstTopElementData REF= stData.stTopElement;

THIS^.refstBaseLoggerElementDataHMI REF= stData.stBaseLoggerElement;
THIS^.refstBaseComponentDataHMI REF= stData.stBaseComponent;
THIS^.refstBaseControlElementDataHMI REF= stData.stBaseControlElement;
THIS^.refstBaseGroupElementDataHMI REF= stData.stBaseGroupElement;
THIS^.refstBaseTopElementDataHMI REF= stData.stBaseTopElement;

THIS^.itfGE1.LinkGroupEData (stData := stData.stGE1);

THIS^.itfCE1.LinkControlEData (stData := stData.stCE1);
THIS^.itfCE2.LinkControlEData (stData := stData.stCE2);

THIS^.itfC1.LinkComponentData (stData := stData.stC1);
THIS^.itfC2.LinkComponentData (stData := stData.stC2);
THIS^.itfC3.LinkComponentData (stData := stData.stC3);

(*
THIS^.itfControlElement1.LinkControlElementData (stData := stData.stControlElement1);
THIS^.itfControlElement2.LinkControlElementData (stData := stData.stControlElement2);
THIS^.itfGroupElement1.LinkGroupelementData (stData := stData.stGroupElement1);
THIS^.itfComponent1.LinkComponentData (stData := stData.stComponent1);
THIS^.itfComponent2.LinkComponentData (stData := stData.stComponent2);
THIS^.itfComponent3.LinkComponentData (stData := stData.stComponent3);
*)
THIS^.CreateLinkToEventsMemory ();

IF (__ISVALIDREF (THIS^.refstTopElementData) AND this^.IsLinkedReferences ()) THEN
	THIS^.bIsValidData		:= TRUE;
	LinkTopElementData		:= TRUE;
END_IF
END_METHOD

END_FUNCTION_BLOCK

// ---- POUs/05_TopElement2/1C_B/FB_Component_TE2.TcPOU
FUNCTION_BLOCK FB_Component_TE2 EXTENDS FB_BaseComponent IMPLEMENTS ITF_Component_TE2, ITF_Component_TE2_HMI_Init
VAR
END_VAR

METHOD testMethod : BOOL
VAR_INPUT
END_VAR
END_METHOD

END_FUNCTION_BLOCK

// ---- POUs/05_TopElement2/2CE_B/FB_ControlE_TE2.TcPOU
FUNCTION_BLOCK FB_ControlE_TE2 EXTENDS FB_BaseControlElement IMPLEMENTS ITF_ControlE_TE2, ITF_ControlE_TE2_HMI_Init
VAR
	itfC1				: ITF_Component_TE2;
	itfC2				: ITF_Component_TE2;
	itfC3				: ITF_Component_TE2;
	itfC4				: ITF_Component_TE2;
	
END_VAR

METHOD FB_init : BOOL
VAR_INPUT
	bInitRetains : BOOL; // if TRUE, the retain variables are initialized (warm start / cold start)
	bInCopyCode : BOOL;  // if TRUE, the instance afterwards gets moved into the copy code (online change)
	itfC1				: ITF_Component_TE2;
	itfC2				: ITF_Component_TE2;
	itfC3				: ITF_Component_TE2;
	itfC4				: ITF_Component_TE2;
END_VAR
THIS^.itfC1 := itfC1;
THIS^.SetText (eLocation := E_BaseLocation.pl, wsDescription := "Komponent 1 EC");
THIS^.SetText (eLocation := E_BaseLocation.en, wsDescription := "Komponent 1 EC");
THIS^.SetText (eLocation := E_BaseLocation.de, wsDescription := "Komponent 1 EC");
itfC1.SetName (stName := THIS^.GetTexts ());
THIS^.AddComponent (itfComponent := itfC1);

THIS^.itfC2 := itfC2;
THIS^.SetText (eLocation := E_BaseLocation.pl, wsDescription := "Komponent 2 EC");
THIS^.SetText (eLocation := E_BaseLocation.en, wsDescription := "Komponent 2 EC");
THIS^.SetText (eLocation := E_BaseLocation.de, wsDescription := "Komponent 2 EC");
itfC2.SetName (stName := THIS^.GetTexts ());
THIS^.AddComponent (itfComponent := itfC2);

THIS^.itfC3 := itfC3;
THIS^.SetText (eLocation := E_BaseLocation.pl, wsDescription := "Komponent 3 EC");
THIS^.SetText (eLocation := E_BaseLocation.en, wsDescription := "Komponent 3 EC");
THIS^.SetText (eLocation := E_BaseLocation.de, wsDescription := "Komponent 3 EC");
itfC3.SetName (stName := THIS^.GetTexts ());
THIS^.AddComponent (itfComponent := itfC3);

THIS^.itfC4 := itfC4;
THIS^.SetText (eLocation := E_BaseLocation.pl, wsDescription := "Komponent 4 EC");
THIS^.SetText (eLocation := E_BaseLocation.en, wsDescription := "Komponent 4 EC");
THIS^.SetText (eLocation := E_BaseLocation.de, wsDescription := "Komponent 4 EC");
itfC4.SetName (stName := THIS^.GetTexts ());
THIS^.AddComponent (itfComponent := itfC4);
END_METHOD

METHOD testMethodCE : BOOL
VAR_INPUT
END_VAR
END_METHOD

END_FUNCTION_BLOCK

// ---- POUs/05_TopElement2/3GE_B/FB_GroupE_TE2.TcPOU
FUNCTION_BLOCK FB_GroupE_TE2 EXTENDS FB_BaseGroupElement IMPLEMENTS ITF_GroupE_TE2, ITF_GroupE_TE2_HMI_Init
VAR
	itfCE1				: ITF_ControlE_TE2;
	itfCE2				: ITF_ControlE_TE2;

	itfC1				: ITF_Component_TE2;
	itfC2				: ITF_Component_TE2;
	itfC3				: ITF_Component_TE2;
	itfC4				: ITF_Component_TE2;
	
END_VAR

METHOD FB_init : BOOL
VAR_INPUT
	bInitRetains : BOOL; // if TRUE, the retain variables are initialized (warm start / cold start)
	bInCopyCode : BOOL;  // if TRUE, the instance afterwards gets moved into the copy code (online change)
	itfCE1				: ITF_ControlE_TE2;
	itfCE2				: ITF_ControlE_TE2;
	itfC1				: ITF_Component_TE2;
	itfC2				: ITF_Component_TE2;
	itfC3				: ITF_Component_TE2;
	itfC4				: ITF_Component_TE2;
END_VAR
THIS^.itfCE1 := itfCE1;
THIS^.SetText (eLocation := E_BaseLocation.pl, wsDescription := "Element 1 EC");
THIS^.SetText (eLocation := E_BaseLocation.en, wsDescription := "Element 1 EC");
THIS^.SetText (eLocation := E_BaseLocation.de, wsDescription := "Element 1 EC");
itfCE1.SetName (stName := THIS^.GetTexts ());
THIS^.AddControlElement (itfControlElement := itfCE1);

THIS^.itfCE2 := itfCE2;
THIS^.SetText (eLocation := E_BaseLocation.pl, wsDescription := "Element 2 EC");
THIS^.SetText (eLocation := E_BaseLocation.en, wsDescription := "Element 2 EC");
THIS^.SetText (eLocation := E_BaseLocation.de, wsDescription := "Element 2 EC");
itfCE2.SetName (stName := THIS^.GetTexts ());
THIS^.AddControlElement (itfControlElement := itfCE2);

THIS^.itfC1 := itfC1;
THIS^.SetText (eLocation := E_BaseLocation.pl, wsDescription := "Komponent 1 EC");
THIS^.SetText (eLocation := E_BaseLocation.en, wsDescription := "Komponent 1 EC");
THIS^.SetText (eLocation := E_BaseLocation.de, wsDescription := "Komponent 1 EC");
itfC1.SetName (stName := THIS^.GetTexts ());
THIS^.AddComponent (itfComponent := itfC1);

THIS^.itfC2 := itfC2;
THIS^.SetText (eLocation := E_BaseLocation.pl, wsDescription := "Komponent 2 EC");
THIS^.SetText (eLocation := E_BaseLocation.en, wsDescription := "Komponent 2 EC");
THIS^.SetText (eLocation := E_BaseLocation.de, wsDescription := "Komponent 2 EC");
itfC2.SetName (stName := THIS^.GetTexts ());
THIS^.AddComponent (itfComponent := itfC2);

THIS^.itfC3 := itfC3;
THIS^.SetText (eLocation := E_BaseLocation.pl, wsDescription := "Komponent 3 EC");
THIS^.SetText (eLocation := E_BaseLocation.en, wsDescription := "Komponent 3 EC");
THIS^.SetText (eLocation := E_BaseLocation.de, wsDescription := "Komponent 3 EC");
itfC3.SetName (stName := THIS^.GetTexts ());
THIS^.AddComponent (itfComponent := itfC3);

THIS^.itfC4 := itfC4;
THIS^.SetText (eLocation := E_BaseLocation.pl, wsDescription := "Komponent 4 EC");
THIS^.SetText (eLocation := E_BaseLocation.en, wsDescription := "Komponent 4 EC");
THIS^.SetText (eLocation := E_BaseLocation.de, wsDescription := "Komponent 4 EC");
itfC4.SetName (stName := THIS^.GetTexts ());
THIS^.AddComponent (itfComponent := itfC4);
END_METHOD

METHOD testMethodGE : BOOL
VAR_INPUT
END_VAR
END_METHOD

END_FUNCTION_BLOCK

// ---- POUs/05_TopElement2/9TE_B/FB_TopElement2.TcPOU
FUNCTION_BLOCK FB_TopElement2 EXTENDS FB_BaseTopElement IMPLEMENTS ITF_TopElement2, ITF_TopElement2_HMI_Init
VAR
	itfGE1				: ITF_GroupE_TE2;

	itfCE1				: ITF_ControlE_TE2;
	itfCE2				: ITF_ControlE_TE2;

	itfC1				: ITF_Component_TE2;
	itfC2				: ITF_Component_TE2;
	itfC3				: ITF_Component_TE2;
END_VAR

METHOD FB_init : BOOL
VAR_INPUT
	bInitRetains : BOOL; // if TRUE, the retain variables are initialized (warm start / cold start)
	bInCopyCode : BOOL;  // if TRUE, the instance afterwards gets moved into the copy code (online change)
	itfGE1				: ITF_GroupE_TE2;
	itfCE1				: ITF_ControlE_TE2;
	itfCE2				: ITF_ControlE_TE2;
	itfC1				: ITF_Component_TE2;
	itfC2				: ITF_Component_TE2;
	itfC3				: ITF_Component_TE2;
END_VAR
THIS^.itfGE1 := itfGE1;
THIS^.SetText (eLocation := E_BaseLocation.pl, wsDescription := "Element złożony 1");
THIS^.SetText (eLocation := E_BaseLocation.en, wsDescription := "Element złożony 1");
THIS^.SetText (eLocation := E_BaseLocation.de, wsDescription := "Element złożony 1");
itfGE1.SetName (stName := THIS^.GetTexts ());
THIS^.AddControlElement (itfControlElement := itfGE1);

THIS^.itfCE1 := itfCE1;
THIS^.SetText (eLocation := E_BaseLocation.pl, wsDescription := "Element wykonawczy 1");
THIS^.SetText (eLocation := E_BaseLocation.en, wsDescription := "Element wykonawczy 1");
THIS^.SetText (eLocation := E_BaseLocation.de, wsDescription := "Element wykonawczy 1");
itfCE1.SetName (stName := THIS^.GetTexts ());
THIS^.AddControlElement (itfControlElement := itfCE1);

THIS^.itfCE2 := itfCE2;
THIS^.SetText (eLocation := E_BaseLocation.pl, wsDescription := "Element wykonawczy 2");
THIS^.SetText (eLocation := E_BaseLocation.en, wsDescription := "Element wykonawczy 2");
THIS^.SetText (eLocation := E_BaseLocation.de, wsDescription := "Element wykonawczy 2");
itfCE2.SetName (stName := THIS^.GetTexts ());
THIS^.AddControlElement (itfControlElement := itfCE2);


THIS^.itfC1 := itfC1;
THIS^.SetText (eLocation := E_BaseLocation.pl, wsDescription := "Komponent 1");
THIS^.SetText (eLocation := E_BaseLocation.en, wsDescription := "Komponent 1");
THIS^.SetText (eLocation := E_BaseLocation.de, wsDescription := "Komponent 1");
itfC1.SetName (stName := THIS^.GetTexts ());
THIS^.AddComponent (itfComponent := itfC1);

THIS^.itfC2 := itfC2;
THIS^.SetText (eLocation := E_BaseLocation.pl, wsDescription := "Komponent 2");
THIS^.SetText (eLocation := E_BaseLocation.en, wsDescription := "Komponent 2");
THIS^.SetText (eLocation := E_BaseLocation.de, wsDescription := "Komponent 2");
itfC2.SetName (stName := THIS^.GetTexts ());
THIS^.AddComponent (itfComponent := itfC2);

THIS^.itfC3 := itfC3;
THIS^.SetText (eLocation := E_BaseLocation.pl, wsDescription := "Komponent 3");
THIS^.SetText (eLocation := E_BaseLocation.en, wsDescription := "Komponent 3");
THIS^.SetText (eLocation := E_BaseLocation.de, wsDescription := "Komponent 3");
itfC3.SetName (stName := THIS^.GetTexts ());
THIS^.AddComponent (itfComponent := itfC3);
END_METHOD

END_FUNCTION_BLOCK

// ---- POUs/05_TopElement2/1C_B_HMI/FB_Component_TE2_HMI.TcPOU
FUNCTION_BLOCK FB_Component_TE2_HMI EXTENDS FB_BaseComponent_HMI IMPLEMENTS ITF_Component_TE2_HMI
VAR
	itfComponent_TE2Connector		: ITF_Component_TE2_HMI_Connector;
	refstComponent_TE2Data			: REFERENCE TO ST_Component_TE2_HMI;

	
END_VAR

METHOD FB_init : BOOL
VAR_INPUT
	bInitRetains : BOOL; // if TRUE, the retain variables are initialized (warm start / cold start)
	bInCopyCode : BOOL;  // if TRUE, the instance afterwards gets moved into the copy code (online change)
	itfBaseLoggerConnector				: ITF_BaseLogger_HMI_Connector;	//bezpośredni łącznik do logera
	itfComponent_TE2Connector			: ITF_Component_TE2_HMI_Init;
END_VAR
//Przypisanie do elementu który własnie stworzyliśmy
THIS^.itfComponent_TE2Connector			:= itfComponent_TE2Connector;
//Przypisanie do elementów z biblioteki
THIS^.itfBaseLoggerElementConnector		:= itfComponent_TE2Connector;
THIS^.itfBaseComponentConnector			:= itfComponent_TE2Connector;

//
THIS^.itfBaseLoggerConnector			:= itfBaseLoggerConnector;

IF (THIS^.itfComponent_TE2Connector <> 0 AND
	THIS^.itfBaseLoggerElementConnector <> 0 AND
	THIS^.itfBaseComponentConnector	<> 0 AND
	THIS^.itfBaseLoggerConnector <> 0) THEN
	THIS^.bIsInit						:= TRUE;
END_IF
END_METHOD

METHOD LinkComponentData : BOOL
VAR_INPUT
	stData				: REFERENCE TO ST_Component_TE2_HMI_Link;
END_VAR
THIS^.refstComponent_TE2Data REF= stData.stComponent_TE2;

THIS^.refstBaseLoggerElementDataHMI REF= stData.stBaseLoggerElement;
THIS^.refstBaseComponentDataHMI REF= stData.stBaseComponent;



THIS^.CreateLinkToEventsMemory ();

IF (__ISVALIDREF (THIS^.refstComponent_TE2Data) AND this^.IsLinkedReferences ()) THEN
	THIS^.bIsValidData		:= TRUE;
	LinkComponentData		:= TRUE;
END_IF
END_METHOD

END_FUNCTION_BLOCK

// ---- POUs/05_TopElement2/2CE_B_HMI/FB_ControlE_TE2_HMI.TcPOU
FUNCTION_BLOCK FB_ControlE_TE2_HMI EXTENDS FB_BaseControlElement_HMI IMPLEMENTS ITF_ControlE_TE2_HMI
VAR
	itfControlE_TE2Connector		: ITF_ControlE_TE2_HMI_Connector;
	refstControlE_TE2Data			: REFERENCE TO ST_ControlE_TE2_HMI;

	itfC1				: ITF_Component_TE2_HMI;
	itfC2				: ITF_Component_TE2_HMI;
	itfC3				: ITF_Component_TE2_HMI;
	itfC4				: ITF_Component_TE2_HMI;
	
END_VAR

METHOD FB_init : BOOL
VAR_INPUT
	bInitRetains : BOOL; // if TRUE, the retain variables are initialized (warm start / cold start)
	bInCopyCode : BOOL;  // if TRUE, the instance afterwards gets moved into the copy code (online change)
	itfBaseLoggerConnector				: ITF_BaseLogger_HMI_Connector;	//bezpośredni łącznik do logera
	itfControlE_TE2Connector			: ITF_ControlE_TE2_HMI_Connector;
	itfC1								: ITF_Component_TE2_HMI;
	itfC2								: ITF_Component_TE2_HMI;
	itfC3								: ITF_Component_TE2_HMI;
	itfC4								: ITF_Component_TE2_HMI;
END_VAR
//Przypisanie do elementu który własnie stworzyliśmy
THIS^.itfControlE_TE2Connector := itfControlE_TE2Connector;
//Przypisanie do elementów z biblioteki
THIS^.itfBaseLoggerElementConnector := itfControlE_TE2Connector;
THIS^.itfBaseComponentConnector := itfControlE_TE2Connector;
THIS^.itfBaseControlElementConnector := itfControlE_TE2Connector;

THIS^.AddComponent (itfComponentHMI := itfC1);
THIS^.itfC1 := itfC1;
THIS^.AddComponent (itfComponentHMI := itfC2);
THIS^.itfC2 := itfC2;
THIS^.AddComponent (itfComponentHMI := itfC3);
THIS^.itfC3 := itfC3;
THIS^.AddComponent (itfComponentHMI := itfC4);
THIS^.itfC4 := itfC4;


//
THIS^.itfBaseLoggerConnector			:= itfBaseLoggerConnector;

IF (THIS^.itfControlE_TE2Connector <> 0 AND
	THIS^.itfBaseLoggerElementConnector <> 0 AND
	THIS^.itfBaseComponentConnector	<> 0 AND
	THIS^.itfBaseControlElementConnector <> 0 AND
	THIS^.itfBaseLoggerConnector <> 0) THEN
	THIS^.bIsInit						:= TRUE;
END_IF
END_METHOD

METHOD LinkControlEData : BOOL
VAR_INPUT
	stData				: REFERENCE TO ST_ControlE_TE2_HMI_Link;
END_VAR
THIS^.refstControlE_TE2Data REF= stData.stControlE_TE2;

THIS^.refstBaseLoggerElementDataHMI REF= stData.stBaseLoggerElement;
THIS^.refstBaseComponentDataHMI REF= stData.stBaseComponent;
THIS^.refstBaseControlElementDataHMI REF= stData.stBaseControlElement;

THIS^.itfC1.LinkComponentData (stData := stData.stComponetE1_TE2);
THIS^.itfC2.LinkComponentData (stData := stData.stComponetE2_TE2);
THIS^.itfC3.LinkComponentData (stData := stData.stComponetE3_TE2);
THIS^.itfC4.LinkComponentData (stData := stData.stComponetE4_TE2);


THIS^.CreateLinkToEventsMemory ();

IF (__ISVALIDREF (THIS^.refstControlE_TE2Data) AND THIS^.IsLinkedReferences ()) THEN
	THIS^.bIsValidData		:= TRUE;
	LinkControlEData		:= TRUE;
END_IF
END_METHOD

END_FUNCTION_BLOCK

// ---- POUs/05_TopElement2/3GE_B_HMI/FB_GroupE_TE2_HMI.TcPOU
FUNCTION_BLOCK FB_GroupE_TE2_HMI EXTENDS FB_BaseGroupElement_HMI IMPLEMENTS ITF_GroupE_TE2_HMI
VAR
	itfGroupE_TE2Connector		: ITF_GroupE_TE2_HMI_Connector;
	refstGroupE_TE2Data			: REFERENCE TO ST_GroupE_TE2_HMI;
	
	itfCE1				: ITF_ControlE_TE2_HMI;
	itfCE2				: ITF_ControlE_TE2_HMI;

	itfC1				: ITF_Component_TE2_HMI;
	itfC2				: ITF_Component_TE2_HMI;
	itfC3				: ITF_Component_TE2_HMI;
	itfC4				: ITF_Component_TE2_HMI;
	
END_VAR

METHOD FB_init : BOOL
VAR_INPUT
	bInitRetains : BOOL; // if TRUE, the retain variables are initialized (warm start / cold start)
	bInCopyCode : BOOL;  // if TRUE, the instance afterwards gets moved into the copy code (online change)
	itfBaseLoggerConnector			: ITF_BaseLogger_HMI_Connector;	//bezpośredni łącznik do logera
	itfGroupE_TE2Connector			: ITF_GroupE_TE2_HMI_Connector;
	itfCE1							: ITF_ControlE_TE2_HMI;
	itfCE2							: ITF_ControlE_TE2_HMI;
	itfC1								: ITF_Component_TE2_HMI;
	itfC2								: ITF_Component_TE2_HMI;
	itfC3								: ITF_Component_TE2_HMI;
	itfC4								: ITF_Component_TE2_HMI;
END_VAR
//Przypisanie do elementu który własnie stworzyliśmy
THIS^.itfGroupE_TE2Connector := itfGroupE_TE2Connector;
//Przypisanie do elementów z biblioteki
THIS^.itfBaseLoggerElementConnector := itfGroupE_TE2Connector;
THIS^.itfBaseComponentConnector := itfGroupE_TE2Connector;
THIS^.itfBaseControlElementConnector := itfGroupE_TE2Connector;
THIS^.itfBaseGroupElementConnector := itfGroupE_TE2Connector;

THIS^.AddControlElement (itfControlElementHMI := itfCE1);
THIS^.itfCE1 := itfCE1;
THIS^.AddControlElement (itfControlElementHMI := itfCE2);
THIS^.itfCE2 := itfCE2;

THIS^.AddComponent (itfComponentHMI := itfC1);
THIS^.itfC1 := itfC1;
THIS^.AddComponent (itfComponentHMI := itfC2);
THIS^.itfC2 := itfC2;
THIS^.AddComponent (itfComponentHMI := itfC3);
THIS^.itfC3 := itfC3;
THIS^.AddComponent (itfComponentHMI := itfC4);
THIS^.itfC4 := itfC4;


//
THIS^.itfBaseLoggerConnector			:= itfBaseLoggerConnector;

IF (THIS^.itfGroupE_TE2Connector <> 0 AND
	THIS^.itfBaseLoggerElementConnector <> 0 AND
	THIS^.itfBaseComponentConnector	<> 0 AND
	THIS^.itfBaseControlElementConnector <> 0 AND
	THIS^.itfBaseGroupElementConnector <> 0 AND
	THIS^.itfBaseLoggerConnector <> 0) THEN
	THIS^.bIsInit						:= TRUE;
END_IF
END_METHOD

METHOD LinkGroupEData : BOOL
VAR_INPUT
	stData				: REFERENCE TO ST_GroupE_TE2_HMI_Link;
END_VAR
THIS^.refstGroupE_TE2Data REF= stData.stGroupE_TE2;

THIS^.refstBaseLoggerElementDataHMI REF= stData.stBaseLoggerElement;
THIS^.refstBaseComponentDataHMI REF= stData.stBaseComponent;
THIS^.refstBaseControlElementDataHMI REF= stData.stBaseControlElement;
THIS^.refstBaseGroupElementDataHMI REF= stData.stBaseGroupElement;

THIS^.itfCE1.LinkControlEData (stData := stData.stControlE1_TE2);
THIS^.itfCE2.LinkControlEData (stData := stData.stControlE2_TE2);

THIS^.itfC1.LinkComponentData (stData := stData.stComponetE1_TE2);
THIS^.itfC2.LinkComponentData (stData := stData.stComponetE2_TE2);
THIS^.itfC3.LinkComponentData (stData := stData.stComponetE3_TE2);
THIS^.itfC4.LinkComponentData (stData := stData.stComponetE4_TE2);


THIS^.CreateLinkToEventsMemory ();

IF (__ISVALIDREF (THIS^.refstGroupE_TE2Data) AND THIS^.IsLinkedReferences ()) THEN
	THIS^.bIsValidData		:= TRUE;
	LinkGroupEData		:= TRUE;
END_IF
END_METHOD

END_FUNCTION_BLOCK

// ---- POUs/05_TopElement2/9TE_B_HMI/FB_TopElement2_HMI.TcPOU
FUNCTION_BLOCK FB_TopElement2_HMI EXTENDS FB_BaseTopElement_HMI IMPLEMENTS ITF_TopElement1_HMI
VAR
	itfTopElementConnector			: ITF_TopElement2_HMI_Connector;
	refstTopElementData				: REFERENCE TO ST_TopElement2_HMI;
	
	itfGE1							: ITF_GroupE_TE2_HMI;
	
	itfCE1							: ITF_ControlE_TE2_HMI;
	itfCE2							: ITF_ControlE_TE2_HMI;
	
	itfC1							: ITF_Component_TE2_HMI;
	itfC2							: ITF_Component_TE2_HMI;
	itfC3							: ITF_Component_TE2_HMI;
END_VAR

METHOD FB_init : BOOL
VAR_INPUT
	bInitRetains : BOOL; // if TRUE, the retain variables are initialized (warm start / cold start)
	bInCopyCode : BOOL;  // if TRUE, the instance afterwards gets moved into the copy code (online change)
	itfBaseLoggerConnector				: ITF_BaseLogger_HMI_Connector;	//bezpośredni łącznik do logera
	itfTopElementConnector				: ITF_TopElement2_HMI_Init;
	itfGE1								: ITF_GroupE_TE2_HMI;
	itfCE1								: ITF_ControlE_TE2_HMI;
	itfCE2								: ITF_ControlE_TE2_HMI;
	itfC1								: ITF_Component_TE2_HMI;
	itfC2								: ITF_Component_TE2_HMI;
	itfC3								: ITF_Component_TE2_HMI;
END_VAR
//Przypisanie do elementu który własnie stworzyliśmy
THIS^.itfTopElementConnector			:= itfTopElementConnector;
//Przypisanie do elementów z biblioteki
THIS^.itfBaseLoggerElementConnector		:= itfTopElementConnector;
THIS^.itfBaseComponentConnector			:= itfTopElementConnector;
THIS^.itfBaseControlElementConnector	:= itfTopElementConnector;
THIS^.itfBaseGroupElementConnector		:= itfTopElementConnector;
THIS^.itfBaseTopElementConnector		:= itfTopElementConnector;
//
THIS^.itfBaseLoggerConnector			:= itfBaseLoggerConnector;

THIS^.AddControlElement (itfControlElementHMI := itfGE1);
THIS^.itfGE1 := itfGE1;

THIS^.AddControlElement (itfControlElementHMI := itfCE1);
THIS^.itfCE1 := itfCE1;

THIS^.AddControlElement (itfControlElementHMI := itfCE2);
THIS^.itfCE2 := itfCE2;

THIS^.AddComponent (itfComponentHMI := itfC1);
THIS^.itfC1 := itfC1;

THIS^.AddComponent (itfComponentHMI := itfC2);
THIS^.itfC2 := itfC2;

THIS^.AddComponent (itfComponentHMI := itfC3);
THIS^.itfC3 := itfC3;

IF (THIS^.itfTopElementConnector <> 0 AND
	THIS^.itfBaseLoggerElementConnector <> 0 AND
	THIS^.itfBaseComponentConnector	<> 0 AND
	THIS^.itfBaseControlElementConnector <> 0 AND
	THIS^.itfBaseGroupElementConnector <> 0 AND
	THIS^.itfBaseTopElementConnector <> 0 AND
	THIS^.itfBaseLoggerConnector <> 0) THEN
	THIS^.bIsInit						:= TRUE;
END_IF
END_METHOD

METHOD LinkTopElementData : BOOL
VAR_INPUT
	stData				: REFERENCE TO ST_TopElement2_HMI_Link;
END_VAR

VAR
	stBaseGroupElem: INT;
END_VAR
THIS^.refstTopElementData REF= stData.stTopElement;

THIS^.refstBaseLoggerElementDataHMI REF= stData.stBaseLoggerElement;
THIS^.refstBaseComponentDataHMI REF= stData.stBaseComponent;
THIS^.refstBaseControlElementDataHMI REF= stData.stBaseControlElement;
THIS^.refstBaseGroupElementDataHMI REF= stData.stBaseGroupElement;
THIS^.refstBaseTopElementDataHMI REF= stData.stBaseTopElement;

THIS^.itfGE1.LinkGroupEData (stData := stData.stGE1);

THIS^.itfCE1.LinkControlEData (stData := stData.stCE1);
THIS^.itfCE2.LinkControlEData (stData := stData.stCE2);

THIS^.itfC1.LinkComponentData (stData := stData.stC1);
THIS^.itfC2.LinkComponentData (stData := stData.stC2);
THIS^.itfC3.LinkComponentData (stData := stData.stC3);

(*
THIS^.itfControlElement1.LinkControlElementData (stData := stData.stControlElement1);
THIS^.itfControlElement2.LinkControlElementData (stData := stData.stControlElement2);
THIS^.itfGroupElement1.LinkGroupelementData (stData := stData.stGroupElement1);
THIS^.itfComponent1.LinkComponentData (stData := stData.stComponent1);
THIS^.itfComponent2.LinkComponentData (stData := stData.stComponent2);
THIS^.itfComponent3.LinkComponentData (stData := stData.stComponent3);
*)
THIS^.CreateLinkToEventsMemory ();

IF (__ISVALIDREF (THIS^.refstTopElementData) AND this^.IsLinkedReferences ()) THEN
	THIS^.bIsValidData		:= TRUE;
	LinkTopElementData		:= TRUE;
END_IF
END_METHOD

END_FUNCTION_BLOCK

// ---- VISUs/MainScreen.TcVIS
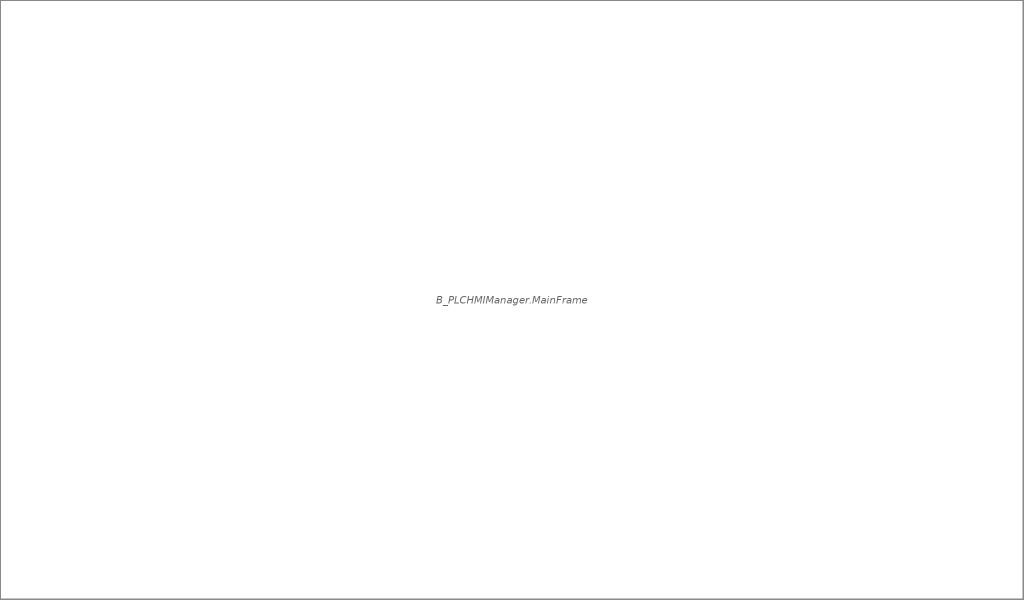
VISUALIZATION MainScreen  // 1024x600
    Frame (0,0 1024x600)
        shows B_PLCHMIManager.MainFrame(stHMIData := PRG_ControlHMI.stHMIData)
END_VISUALIZATION
